# B&R Automation Studio project x20ost (part 4)

#### bnrmytimer.c
```c
/********************************************************************
 * COPYRIGHT -- Kontora
 ********************************************************************
 * Program: bnrmain
 * File: bnrlsens.c
 * Author: Abramenya
 * Created: January 19, 2009
 *******************************************************************/

#include "bnrmytimer.h"
#ifdef _DEFAULT_INCLUDES
 #include <AsDefault.h>
#endif
void CMTimer_OfTimer(This)
{
     DECLARE_MULTI_OPEN(CMTimer,CSystemTimer)
     pB->OfTimer(pB);
}
void CMTimer_OnTimer(This,DWORD dwTime)
{
     DECLARE_MULTI_OPEN(CMTimer,CSystemTimer)
	 pB->OnTimer(pB,dwTime);
	 pT->m_dwSTime = dwTime;
}
void CMTimer_Restart(This)
{
	 DECLARE_MULTI_OPEN(CMTimer,CSystemTimer)
	 pB->OnTimer(pB,pT->m_dwSTime);
}
DWORD CMTimer_GetTime(This)
{
	DECLARE_MULTI_OPEN(CMTimer,CSystemTimer)
	//if pB->m_dwTime
    return pB->m_dwTime;
}
void CMTimer_SetTimer(This,BYTE byFor,BYTE byFrom,BYTE byEvent,BYTE byDir,BYTE bySens,BYTE byBox)
{
     DECLARE_MULTI_OPEN(CMTimer,CSystemTimer)
	 pT->m_byFor   = byFor;
	 pT->m_byFrom  = byFrom;
	 pT->m_byEvent = byEvent;
	 pT->m_byDir   = byDir;
	 pT->m_bySens  = bySens;
	 pT->m_byBox   = byBox;
}
void CMTimer_DoAction(This)
{
	 DECLARE_MULTI_OPEN(CMTimer,CSystemTimer)
	 pT->sMsg.m_swLen        = 9;
	 pT->sMsg.m_sbyFrom      = pT->m_byFrom;
	 pT->sMsg.m_sbyFor       = pT->m_byFor;
	 pT->sMsg.m_sbyIntType   = 0;
	 pT->sMsg.m_sbyServerID  = MYSYSTEM_ID;
	 pT->sMsg.m_sbyDirection = pT->m_byDir;
	 pT->sMsg.m_sbySensor    = pT->m_bySens;
	 pT->sMsg.m_sbyType      = pT->m_byEvent;
	 FPUT(pT->m_byBox,(BYTE*)&pT->sMsg);
}
void CMTimer_CMTimer(This)
{
     DECLARE_MULTI_OPEN(CMTimer,CSystemTimer)
	 DECLARE_REGISTRATION(CMTimer,GetTime)
	 DECLARE_REGISTRATION(CMTimer,OnTimer)
	 DECLARE_REGISTRATION(CMTimer,OfTimer)
	 DECLARE_REGISTRATION(CMTimer,SetTimer)
	 DECLARE_REGISTRATION(CMTimer,Restart)
	 DECLARE_VIRTUAL_FUNC(CMTimer,DoAction)
}
void CMTimer_DCMTimer(This)
{
	 DECLARE_MULTI_OPEN(CMTimer,CSystemTimer)
}
DECLARE_MULTI_CREATE(CMTimer,CSystemTimer)
```

#### bnrobserve.c
```c
/********************************************************************
 * COPYRIGHT -- Kontora
 ********************************************************************
 * Program: bnrmain
 * File: bnrlsens.c
 * Author: Abramenya
 * Created: January 19, 2009
 *******************************************************************/

#include "bnrobserve.h"
#if MYSYSTEM_ID != 5
#ifdef _DEFAULT_INCLUDES
#include <AsDefault.h>
#endif
CObserveModule *pvOBS;
_GLOBAL PFNVOID pfnAnalogDataReq;
_GLOBAL PFNVOID pfnDigitalDataReq;
void AnalogDataReq(void);
void DigitalDataReq(void);
void CObserveModule_Init(This,SSOFTSWITCHTABLE *pSoftSwitchTable)
{
    DECLARE_MULTI_OPEN(CObserveModule,CCyclicSystem)
	pvOBS = pT;
	pfnAnalogDataReq  = AnalogDataReq;
    pfnDigitalDataReq = DigitalDataReq;
	pT->m_byTableVersion = pSoftSwitchTable->byTableVersion;
	strcpy(pT->m_chTableVersionName,pSoftSwitchTable->chTableVersionName);
	pT->m_byAmDirection = pSoftSwitchTable->byAmDirection;
    //#ifdef DEB_CObserveModule
	Info("\n(__)COBSE::>Create Observation Module: %s",pSoftSwitchTable->chTableVersionName);
    //#endif
    pT->CreateObserve(pT,pSoftSwitchTable);
	pT->m_byObsTime = T2SEC;
	InitObject(CMTimer,&pT->m_pRefrechTmr);
	pT->m_pRefrechTmr.SetTimer(&pT->m_pRefrechTmr,MDL_OBSRV,MDL_OBSRV,EV_OBSRV_REFR_TIM_PROC_IND,0,0,DEV_SYSTM_BOX_ID);
}
_GLOBAL INT iCObserveModuleVal;
void CObserveModule_CreateObserve(This,SSOFTSWITCHTABLE *pSoftSwitchTable)
{
    DECLARE_MULTI_OPEN(CObserveModule,CCyclicSystem)
	CDirectionModule *p;
	INT i;
	InitObject(CMFlash,&pT->m_nFlash);
	pT->m_byAmDirection = pSoftSwitchTable->byAmDirection;
	New(sizeof(CDirectionModule*)*pT->m_byAmDirection,pT->m_pDirectionModule);
	for(i=0;i<pT->m_byAmDirection;i++)
	{
	 New(sizeof(CDirectionModule),p);
	 InitObject(CDirectionModule,p);
	 if(p!=NULL)
	 {
	  iCObserveModuleVal++;
	  p->ConnectToComputer(p,pT->m_pComputer);
      p->ConnectToAdmin(p,pT->m_pAdmin);
	  p->m_bySystemID = pT->m_bySystemID;
	  p->Init(p,&pSoftSwitchTable->sDirectionTable[i],&pT->m_nFlash);
	  pT->m_pDirectionModule[i] = p;
	 }
	}
}
void CObserveModule_SetSystemID(This,BYTE bySystemID)
{
     DECLARE_MULTI_OPEN(CObserveModule,CCyclicSystem)
     pT->m_bySystemID = bySystemID;
}
void CObserveModule_ConnectToAdmin(This,CAdmin *pAdmin)
{
     DECLARE_MULTI_OPEN(CObserveModule,CCyclicSystem)
	 pT->m_pAdmin = pAdmin;
}
//_GLOBAL INT nVAL_0;
BOOL CObserveModule_EventHandler(This,SMESSAGE *pMsg)
{
	 BOOL res = TRUE;
     DECLARE_MULTI_OPEN(CObserveModule,CCyclicSystem)
	 CDirectionModule *pD;SPIN sP;CSensor *pS;
	 WORD wValue,wValue1; BYTE byValue,*pBT;
	 #ifdef DEB_CObserveModule
	 if(dwFL&DEB_OUT_OBSR_COMM)
	 Info("\n(%b)COBSE::>MSG::%M",&pT->m_bySystemID,(BYTE*)pMsg);
     #endif
     switch (pMsg->m_sbyFor)
	 {
		case MDL_OBSRV:
             switch (pMsg->m_sbyType)
			 {
                case EV_OBSRV_GET_MODE_REQ: //Запросить выходное состояние сенсоров направления	140
                     if((pD=pT->GetDirection(pT,pMsg->m_sbyDirection))!=0)
					 {
					 pD->GetDirMode(pD,pMsg);
					 #ifdef DEB_CObserveModule
					 if(dwFL&DEB_OUT_OBSR_COMM)
					 Info("\n(%b)COBSE::>DC(%b,X)SET_MODE",&pT->m_bySystemID,&pMsg->m_sbyDirection);
                     #endif
					 }
     	        break;
				case EV_OBSRV_SET_MODE_REQ:
					 if((pD=pT->GetDirection(pT,pMsg->m_sbyDirection))!=0)
					 {
					 pD->SetDirMode(pD,pMsg);
                     #ifdef DEB_CObserveModule
					 if(dwFL&DEB_OUT_OBSR_COMM)
					 Info("\n(%b)COBSE::>DC(%b,X)SET_MODE",&pT->m_bySystemID,&pMsg->m_sbyDirection);
                     #endif
					 }
				break;
				case EV_OBSRV_START_DATA_PROC_REQ:
					 byValue = pMsg->m_sbyInfo[1];
					 pT->m_byObserveProc = pMsg->m_sbyInfo[2];
                     pT->m_byObsTime = byValue;
                     pT->m_pRefrechTmr.OnTimer(&pT->m_pRefrechTmr,pT->m_byObsTime);
					 //pT->m_pRefrechTmr.OnTimer(&pT->m_pRefrechTmr,10);
                     //#ifdef DEB_CObserveModule
					 //if(dwFL&DEB_OUT_OBSR_COMM)
					 //Info("\n(%b)COBSE::>DC(%b,X)START_DATA_PROC_REQ:[%b]:[%b]",&pT->m_bySystemID,&pMsg->m_sbyDirection,&byValue,&pT->m_byObserveProc);
                     //#endif
				break;
				case EV_OBSRV_STOP_DATA_PROC_REQ:
					 pT->m_pRefrechTmr.OfTimer(&pT->m_pRefrechTmr);
                     #ifdef DEB_CObserveModule
					 if(dwFL&DEB_OUT_OBSR_COMM)
					 Info("\n(%b)COBSE::>DC(%b,X)STOP_DATA_PROC_REQ",&pT->m_bySystemID,&pMsg->m_sbyDirection);
                     #endif
				break;
                case EV_OBSRV_REFR_TIM_PROC_IND: //Таймер обновления данных
					 if(pT->m_byObserveProc==0)pT->GetObserveData(pT,EV_OBSRV_GET_OUT_DATA_IND);
					 if(pT->m_byObserveProc==1)pT->GetObserveData(pT,EV_OBSRV_GET_DMC_DATA_IND);
					 //if(pT->m_byObserveProc==0)pfnAnalogDataReq();
					 //if(pT->m_byObserveProc==1)pfnDigitalDataReq();
					 pT->m_pRefrechTmr.OnTimer(&pT->m_pRefrechTmr,pT->m_byObsTime);
					 //pT->m_pRefrechTmr.OnTimer(&pT->m_pRefrechTmr,10);
                     #ifdef DEB_CObserveModule
					 if(dwFL&DEB_OUT_OBSR_COMM)
					 Info("\n(%b)COBSE::>DC(%b,X)GET_INOUT_SDATA_IND",&pT->m_bySystemID,&pMsg->m_sbyDirection);
                     #endif
				break;
				case EV_OBSRV_RFLASH_SAVE_REQ:
				     //nVAL_0++;
					 pT->m_pDirectionModule[0]->m_byDefSett = 0;
			         pT->m_pDirectionModule[0]->Serialize(pT->m_pDirectionModule[0],TRUE);
				break;
                default:
		        break;
			 }
		break;
		case MDL_PSENS://Digital Sensor
			 if((pS=pT->GetSensor(pT,&pD,pMsg->m_sbyDirection,pMsg->m_sbySensor))!=0)
			 pS->EventHandler(pS->pChld,pMsg);
		break;
        #if MYSYSTEM_ID !=4
		case MDL_SENSR:
			 if((pS=pT->GetSensor(pT,&pD,pMsg->m_sbyDirection,pMsg->m_sbySensor))!=0)
			 pS->SEventHandler(pS,pMsg);
		break;
		case MDL_SSENS:
			 if((pS=pT->GetSensor(pT,&pD,pMsg->m_sbyDirection,pMsg->m_sbySensor))!=0)
	         pS->EventHandler(pS->pChld,pMsg);
		break;
        #endif
		case MDL_DIRMD:
			 if((pD=pT->GetDirection(pT,pMsg->m_sbyDirection))!=0)
			 pD->EventHandler(pD,pMsg);
		break;
		default:
		break;
	};
	return res;
}
//_GLOBAL INT nAnData;
void AnalogDataReq(void)
{
	pvOBS->GetObserveData(pvOBS,EV_OBSRV_GET_OUT_DATA_IND);
	//nAnData++;
}
void DigitalDataReq(void)
{
    pvOBS->GetObserveData(pvOBS,EV_OBSRV_GET_DMC_DATA_IND);
}
void CObserveModule_GetObserveData(This,BYTE byEvent)
{
	DECLARE_MULTI_OPEN(CObserveModule,CCyclicSystem)
	INT i,j=0;
	CDirectionModule *p;
	SMESSAGE *pM = &pT->m_nMsg;
	BYTE *pMB = &pM->m_sbyInfo[0];
	pM->m_sbyFrom      = MDL_OBSRV;
	pM->m_sbyFor       = MDL_ARMSY;
	pM->m_sbyIntType   = DEV_ARM_PORT_TCP;
	pM->m_sbyType      = byEvent;
	pM->m_sbyServerID  = pT->m_bySystemID;
	pM->m_sbySensor    = 0xff;
	pM->m_swLen        = 9;
	for(i=0;i<pT->m_byAmDirection;i++)
	{
	 p = pT->m_pDirectionModule[i];
	 if(byEvent==EV_OBSRV_GET_OUT_DATA_IND)j = p->GetXWData(p,(SMESSAGE*)&pMB[j]);
	 if(byEvent==EV_OBSRV_GET_DMC_DATA_IND)j = p->GetDigMcData(p,(SMESSAGE*)&pMB[j]);
	 pM->m_swLen += j;
	 //Info("\n(%b)COBSE::>Put:%w",&pT->m_bySystemID,&pM->m_swLen);
	}
	pM->m_sbyDirection = pT->m_byAmDirection;
	if(pT->m_pAdmin->m_blArmState)
	FPUT(DEV_ARMOT_BOX_ID,(BYTE*)pM);
	if(dwFL&DEB_OUT_OBSR_COMM)
	Info("\n(%b)COBSE::>MSG:%M",&pT->m_bySystemID,(BYTE*)pM);
}
CDirectionModule* CObserveModule_GetDirection(This,BYTE byDir)
{
	DECLARE_MULTI_OPEN(CObserveModule,CCyclicSystem)
	CDirectionModule *pD;
	if(byDir<pT->m_byAmDirection)
		return pD = pT->m_pDirectionModule[byDir];
	return 0;
}
CSensor* CObserveModule_GetSensor(This,CDirectionModule **pD,BYTE byDir,BYTE bySensor)
{
	DECLARE_MULTI_OPEN(CObserveModule,CCyclicSystem)
	CDirectionModule *pDM = *pD;
	if(byDir<pT->m_byAmDirection)
	{
	 pDM = pT->m_pDirectionModule[byDir];
	 *pD = pDM;
	 if(bySensor < pDM->m_byAmSwitching)
	 return pDM->m_pSensor[bySensor];
	}
	return 0;
}
void CObserveModule_CyclicProc(This)
{
	DECLARE_MULTI_OPEN(CObserveModule,CCyclicSystem)
	CDirectionModule *p;INT i;
    for(i=0;i<pT->m_byAmDirection;i++)
	{
	  p = pT->m_pDirectionModule[i];
	  p->ObserveProc(p);
	}
}
void CObserveModule_ConnectToComputer(This,CComputer *pComputer)
{
    DECLARE_MULTI_OPEN(CObserveModule,CCyclicSystem)
	pT->m_pComputer = pComputer;
}
void CObserveModule_CObserveModule(This)
{
    DECLARE_MULTI_OPEN(CObserveModule,CCyclicSystem)
	DECLARE_REGISTRATION(CObserveModule,Init)
	DECLARE_REGISTRATION(CObserveModule,ConnectToComputer)
	DECLARE_REGISTRATION(CObserveModule,CreateObserve)
	DECLARE_REGISTRATION(CObserveModule,GetObserveData)
	DECLARE_REGISTRATION(CObserveModule,SetSystemID)
	DECLARE_REGISTRATION(CObserveModule,GetDirection)
	DECLARE_REGISTRATION(CObserveModule,GetSensor)
	DECLARE_REGISTRATION(CObserveModule,SetSystemID)
	DECLARE_REGISTRATION(CObserveModule,ConnectToAdmin)
	DECLARE_VIRTUAL_FUNC(CObserveModule,EventHandler)
	DECLARE_VIRTUAL_FUNC(CObserveModule,CyclicProc)
}
void CObserveModule_DCObserveModule(This)
{
	DECLARE_MULTI_OPEN(CObserveModule,CCyclicSystem)
	BYTE i;
	for(i=0;i<pT->m_byAmDirection;i++)
	DestroyObject(CDirectionModule,pT->m_pDirectionModule[i]);
	Delete(sizeof(CDirectionModule*)*pT->m_byAmDirection,pT->m_pDirectionModule);
}
DECLARE_MULTI_CREATE(CObserveModule,CCyclicSystem)
#endif
```

#### bnroutgate.c
```c
/********************************************************************
 * COPYRIGHT -- Kontora
 ********************************************************************
 * Program: bnrmain
 * File: bnrlsens.c
 * Author: Abramenya
 * Created: January 19, 2009
 *******************************************************************/

#include "bnroutgate.h"
#ifdef _DEFAULT_INCLUDES
 #include <AsDefault.h>
#endif
#if MYSYSTEM_ID != 5
void COutGate_Init(This,BYTE byID,BYTE byType,BYTE byOType,BYTE byMode,REAL rMinRamp,REAL rMaxRamp,CPin *pPin,UINT wLo,UINT wHi,UINT wIni,BYTE byState,WORD wBase,WORD wOTime,SINT *pName)
{
    DECLARE_SINGLE_OPEN(COutGate)
	REAL rHL        = (REAL)(wHi-wLo);
	REAL rIP        = (REAL)wIni;
	pT->m_rMinRamp  = rMinRamp;
	pT->m_rMaxRamp  = rMaxRamp;
	pT->m_wBase     = wBase;
	pT->m_byState   = byState;
	pT->m_byGateID  = byID;
	pT->m_byType    = byType;
	pT->m_byOType   = byOType;  //BASE_GTE
	pT->m_byMode    = byMode;
	pT->m_wQTime    = SYSTEM_QTIME;
	pT->m_wLoLimit  = 0;
	pT->m_wHiLimit  = wHi-wLo;
    pT->m_wIniState = (UINT)(rHL*rIP/100.0);
	pT->m_wCurrOpenState = pT->m_wIniState;
	pT->m_dwTime    = 0;
	pT->m_pConnectionPin = pPin;
	if(pPin!=0)pT->m_pwOut = (UINT*)pPin->GetAddrPin(pPin->pChld); else
	pT->m_pwOut = &pT->m_wOut;
	pT->m_wTick     = 0;
	pT->m_wOTime = wOTime;
	if(pT->m_wOTime==0) pT->m_wOTime=1;
	pT->m_wMaxQt = (REAL)pT->m_wOTime*10;
	pT->m_wTickConst = (REAL)pT->m_wHiLimit/pT->m_wMaxQt;
    pT->m_wTickOpen  = pT->m_wTickConst;
	pT->m_blProccState = FALSE;
	pT->m_wMinRampValue = (UINT)(rHL*pT->m_rMinRamp);
	pT->m_wMaxRampValue = (UINT)(rHL*pT->m_rMaxRamp);

	strcpy(pT->m_chName,pName);
}
void COutGate_SetOutTime(This,WORD wValue)
{
    DECLARE_SINGLE_OPEN(COutGate)
	pT->m_wMaxQt = (REAL)wValue*10;
	if(pT->m_wMaxQt==0)return;
    pT->m_wTickConst = pT->m_wHiLimit/pT->m_wMaxQt;
	pT->m_wTickOpen  = pT->m_wTickConst;
}
void COutGate_SetHiLimit(This,WORD wValue)
{
    DECLARE_SINGLE_OPEN(COutGate)
    pT->m_wHiLimit = wValue;
	pT->m_wTickConst = pT->m_wHiLimit/pT->m_wMaxQt;
    pT->m_wTickOpen  = pT->m_wTickConst;
}
//UINT _GLOBAL nmMaxRamp,nOutVal,nMinR,nMaxR,nCOpen;
//REAL _GLOBAL rgValue,rHILM,rMaxRamp;
void COutGate_SetMinRamp(This,REAL rValue)
{
    DECLARE_SINGLE_OPEN(COutGate)
	REAL rMaxValue = (REAL)pT->m_wHiLimit;
    pT->m_rMinRamp = rValue;
	pT->m_wMinRampValue = (UINT)(rMaxValue*pT->m_rMinRamp);
}
void COutGate_SetMaxRamp(This,REAL rValue)
{
    DECLARE_SINGLE_OPEN(COutGate)
	REAL rMaxValue = (REAL)pT->m_wHiLimit;
	pT->m_rMaxRamp = rValue;
	pT->m_wMaxRampValue = (UINT)(rMaxValue*pT->m_rMaxRamp);

	//nmMaxRamp = pT->m_wHiLimit;
	//rHILM     = rMaxValue;
	//rgValue   = rValue;
	//rMaxRamp  = pT->m_wMaxRampValue;
}
void COutGate_OpenGate(This,REAL rOpenState)
{
    DECLARE_SINGLE_OPEN(COutGate)
	UINT wEndState;
	REAL rHi;
	//if(!pT->m_blProccState)
	{
	 rHi = (REAL)pT->m_wHiLimit;
	 wEndState = (UINT)(rOpenState*rHi/100.0);
	 if (wEndState==pT->m_wCurrOpenState) return;
	 pT->m_wTickOpen = pT->m_wTickConst;
	 if (wEndState < pT->m_wCurrOpenState)
     pT->m_wTickOpen = -pT->m_wTickConst;
     pT->m_wTick = (DWORD)(abs(pT->m_wCurrOpenState-wEndState)/pT->m_wTickConst);
	 pT->m_wOperGate = (REAL)pT->m_wCurrOpenState;
	 pT->m_blProccState = TRUE;
	};
}
void COutGate_OpenGateReq(This,BYTE byOpenState)
{
    DECLARE_SINGLE_OPEN(COutGate)
	UINT wEndState;
	REAL rHi;
	if (byOpenState<=100)
	{
	 rHi = (REAL)pT->m_wHiLimit;
     wEndState = (UINT)((REAL)byOpenState*rHi/100.0);
	 pT->SetManGate(pT,wEndState);
	}
}
void COutGate_StopGate(This)
{
    DECLARE_SINGLE_OPEN(COutGate)
    pT->m_blProccState = FALSE;
	pT->m_wTick = 0;
}
void COutGate_SetGate(This,UINT wValue)
{
	DECLARE_SINGLE_OPEN(COutGate)
	//nOutVal = wValue;
	//nMinR   = pT->m_wMinRampValue;
	//nMaxR   = pT->m_wMaxRampValue;
	if (wValue<pT->m_wMinRampValue) wValue = pT->m_wMinRampValue;
	if (wValue>pT->m_wMaxRampValue) wValue = pT->m_wMaxRampValue;
	//if((wValue>=pT->m_wMinRampValue)&&(wValue<=pT->m_wMaxRampValue+20))
	//{
	pT->m_wCurrOpenState = wValue;
	//nCOpen = wValue;
    if(pT->m_byState==ST_OPEN)
	{
	 if(pT->m_byOType==NZ) *pT->m_pwOut = pT->m_wBase+pT->m_wCurrOpenState;
	 if(pT->m_byOType==NO) *pT->m_pwOut = pT->m_wBase+(pT->m_wHiLimit-pT->m_wCurrOpenState);
	}
	//}
}
void COutGate_SetManGate(This,UINT wValue)
{
	DECLARE_SINGLE_OPEN(COutGate)
	pT->m_wCurrOpenState = wValue;
    if(pT->m_byState==ST_OPEN)
	{
	 if(pT->m_byOType==NZ) *pT->m_pwOut = pT->m_wBase+pT->m_wCurrOpenState;
	 if(pT->m_byOType==NO) *pT->m_pwOut = pT->m_wBase+(pT->m_wHiLimit-pT->m_wCurrOpenState);
	}
}
UINT COutGate_GetGate(This)
{
	DECLARE_SINGLE_OPEN(COutGate)
	if(pT->m_byOType==NZ)return pT->m_wBase+pT->m_wCurrOpenState;
	if(pT->m_byOType==NO)return pT->m_wBase+(pT->m_wHiLimit-pT->m_wCurrOpenState);
	return 0;
}
BYTE COutGate_GetPrcGate(This)
{
	DECLARE_SINGLE_OPEN(COutGate)
	//REAL rC = pT->m_wCurrOpenState;
	//REAL rH = pT->m_wHiLimit;
	//return (BYTE)(100.0*rC/rH);
	return (BYTE)(100.0*pT->m_wCurrOpenState/pT->m_wHiLimit);
	//return (BYTE)(100.0*pT->m_wCurrOpenState/6683.0);
}
void COutGate_RunGate(This)
{
    DECLARE_SINGLE_OPEN(COutGate)
	if(pT->m_blProccState)
	{
	 if(pT->m_wTick!=0)
	 {
	  pT->m_wOperGate += pT->m_wTickOpen;
	  //Info("\n(__)Tick:%b Val:%w",&pT->m_wTick,&pT->m_wCurrOpenState.iValue);
	  pT->SetManGate(pT,(UINT)pT->m_wOperGate);
	  pT->m_wTick--;
	 }else pT->m_blProccState = FALSE;
	}
}
void COutGate_SetDefault(This)
{
    DECLARE_SINGLE_OPEN(COutGate)
	pT->SetGate(pT,pT->m_wIniState);
}
void COutGate_SetState(This,BYTE byState)
{
    DECLARE_SINGLE_OPEN(COutGate)
	if(byState==ST_INIT)pT->SetDefault(pT);
	pT->m_byState = byState;
}
void COutGate_COutGate(This)
{
    DECLARE_SINGLE_OPEN(COutGate)
	DECLARE_REGISTRATION(COutGate,Init)
	DECLARE_REGISTRATION(COutGate,OpenGate)
    DECLARE_REGISTRATION(COutGate,SetGate)
	DECLARE_REGISTRATION(COutGate,GetGate)
	DECLARE_REGISTRATION(COutGate,RunGate)
	DECLARE_REGISTRATION(COutGate,SetDefault)
	DECLARE_REGISTRATION(COutGate,SetState)
	DECLARE_REGISTRATION(COutGate,GetPrcGate)
	DECLARE_REGISTRATION(COutGate,SetMinRamp)
	DECLARE_REGISTRATION(COutGate,SetMaxRamp)
	DECLARE_REGISTRATION(COutGate,SetHiLimit)
	DECLARE_REGISTRATION(COutGate,SetManGate)
	DECLARE_REGISTRATION(COutGate,StopGate)
	DECLARE_REGISTRATION(COutGate,SetOutTime)
	DECLARE_REGISTRATION(COutGate,OpenGateReq)
}
void COutGate_DCOutGate(This)
{
	DECLARE_SINGLE_OPEN(COutGate)
}
DECLARE_SINGLE_CREATE(COutGate)
#endif
```

#### bnrpin.c
```c
/********************************************************************
 * COPYRIGHT -- Kontora
 ********************************************************************
 * Program: bnrmain
 * File: bnrlsens.c
 * Author: Abramenya
 * Created: January 19, 2009
 *******************************************************************/

#include "bnrpin.h"
#ifdef _DEFAULT_INCLUDES
 #include <AsDefault.h>
#endif
#ifdef DEB_CPin
SINT *chPinState[] =
{
	"DEF",
	"ONN",
	"OFF",
	"TRI",
};
SINT *chPinType[] =
{
	"DEFAULT_PIN",
	"AN_INOT_INT",
	"DG_INOT_BOL",
	"ST_INPT_USI",
	"ST_OUTP_USI"
};
#endif
void CPin_Init(This,SHARDPIN*pPin,SHARDPIN *pAlPin)
{
    DECLARE_SINGLE_OPEN(CPin)
	pT->m_pvAlmState  = pAlPin->pvValue;
	pT->m_byPinState  = pPin->byPinState;
	pT->m_byPinNumber = pPin->byPinNumber;
	pT->InitPin(pC,pPin->pvValue);
	pT->m_blPinON  = FALSE;
	pT->m_blPinOFF = FALSE;
    #ifdef DEB_CPin
	Info("\n(%b)CPINS::>Create Pin: State:[%s] Type:[%s]",&pPin->byPinNumber,chPinState[pPin->byPinState],chPinType[pPin->byPinType]);
    #endif
}

void CPin_SetSlot(This,BYTE bySlot)
{
	DECLARE_SINGLE_OPEN(CPin)
    pT->m_bySlotNumber = bySlot;
}
PVOID CPin_GetAddrPin(This)
{
	DECLARE_SINGLE_OPEN(CPin)
	return 0;
}
BYTE CPin_GetState(This)
{
    DECLARE_SINGLE_OPEN(CPin)
	SPIN sP;
	pT->GetPin(pC,&sP);
	if(sP.blValue)
	{
	 if(pT->m_blPinON==FALSE)
	 {
	  pT->m_blPinON = TRUE;
	  pT->m_blPinOFF= FALSE;
	  return PIN_STATE_ONN;
	 }else return PIN_STATE_TRI;
	}else
	{
	 if(pT->m_blPinOFF==FALSE)
	 {
	  pT->m_blPinOFF= TRUE;
	  pT->m_blPinON = FALSE;
	  return PIN_STATE_OFF;
	 }else return PIN_STATE_TRI;
	}
}
void CPin_GetPin(This,SPIN *sP)
{
    DECLARE_SINGLE_OPEN(CPin)
}
void CPin_CPin(This)
{
    DECLARE_SINGLE_OPEN(CPin)
	DECLARE_REGISTRATION(CPin,Init)
	DECLARE_REGISTRATION(CPin,SetSlot)
	DECLARE_REGISTRATION(CPin,GetAddrPin)
	DECLARE_REGISTRATION(CPin,GetPin)
	DECLARE_REGISTRATION(CPin,GetState)
}
void CPin_DCPin(This)
{
	DECLARE_SINGLE_OPEN(CPin)
}
DECLARE_SINGLE_CREATE(CPin)
```

#### bnrpob.c
```c
#include "bnrpob.h"
#include "bnrmessage.h"
#ifndef WIN32
_GLOBAL pBOX pBufferHiLev[MAXNAMEBUF];
_GLOBAL pBOX nMirrorBuffer;
_GLOBAL BOOL blSMB;
#else
pBOX pBufferHiLev[MAXNAMEBUF];
pBOX nMirrorBuffer;
BOOL blSMB;
#endif
void FFREE(BYTE b_lNmBox)
{
	pBOX *p;
	if(b_lNmBox>MAXNAMEBUF) return;
	nMirrorBuffer.pb_mBoxCont = 0;
	nMirrorBuffer.w_mBoxMesCt = 1;
	blSMB = FALSE;
	p = &pBufferHiLev[b_lNmBox];
	p->w_mBoxSize  = p->w_mBoxCSize;
    p->w_mBoxWrite = 0;
    p->w_mBoxRead  = 0;
    p->w_mBoxMesCt = 0;
}
void FINIT(void)
{
	//BYTE i;
	//for(i=0;i<MAXNAMEBUF-1;i++)pBufferHiLev[i].pb_mBoxCont = 1;
}
int FDEFINE(BYTE b_lNmBox,WORD w_lBoxSize)
{
	pBOX *p;
    if(b_lNmBox>MAXNAMEBUF) return NULL;
	p = &pBufferHiLev[b_lNmBox];
	//if(p->pb_mBoxCont!=1) return b_lNmBox;
	New(sizeof(BYTE)*(w_lBoxSize+BOX_TRANS_SIZE),p->pb_mBoxCont);
    if(p==NULL) return NULL;
	p->w_mBoxSize  = w_lBoxSize;
    p->w_mBoxCSize = w_lBoxSize;
    p->w_mBoxWrite = 0;
    p->w_mBoxRead  = 0;
    p->w_mBoxMesCt = 0;
    #ifdef DEF_CRT_BOX
	Info("\n(%b)CSBOX::>Create System Box.Size:%w",&b_lNmBox,&pBufferHiLev[b_lNmBox]->w_mBoxCSize);
    //Info("\n(%b)CRT:BOX:>:AD[%a]:WR[%w]:RD[%w]:SZ[%w]:CT[%w]",&b_lNmBox,&p,&p->w_mBoxWrite,&p->w_mBoxRead,&p->w_mBoxSize,&p->w_mBoxMesCt);
    #endif
    return 1;
}
void FDELETE(BYTE b_lNmBox)
{
	pBOX *p;
	p = &pBufferHiLev[b_lNmBox];
    Delete(p->w_mBoxCSize+BOX_TRANS_SIZE,p->pb_mBoxCont);
    p->pb_mBoxCont = 0;
    #ifdef DEF_CRT_BOX
    Info("\n(%b)DEL:BOX",&b_lNmBox);
    #endif
}
int FCHECK(BYTE b_lNmBox)
{
    return pBufferHiLev[b_lNmBox].w_mBoxMesCt;
}
int FCHECKM(BYTE b_lNmBox)
{
	if(!blSMB)
	{
	 memcpy(&nMirrorBuffer,&pBufferHiLev[b_lNmBox],sizeof(pBOX));
	 blSMB = TRUE;
	}
    return nMirrorBuffer.w_mBoxMesCt;
}
int FPUT(BYTE b_lNmBox,BYTE *pb_lInBox)
{
	pBOX *p;
    WORD w_lLength;
	p = &pBufferHiLev[b_lNmBox];
    w_lLength = *(WORD*)pb_lInBox;
    if(!p->pb_mBoxCont)return 0;
    if((w_lLength>p->w_mBoxSize)||(w_lLength<2))return 0;
	memcpy(&p->pb_mBoxCont[p->w_mBoxWrite],pb_lInBox,w_lLength);
    p->w_mBoxWrite += w_lLength;
    p->w_mBoxSize  -= w_lLength;
    p->w_mBoxMesCt ++;
    if(p->w_mBoxWrite>p->w_mBoxCSize) p->w_mBoxWrite = 0;
    #ifdef DEF_INF_BOX
    Info("\n(%b)PUTB:>:LN[%w]:WR[%w]:RD[%w]:SZ[%w]:CT[%w]",&b_lNmBox,&w_lLength,&p->w_mBoxWrite,&p->w_mBoxRead,&p->w_mBoxSize,&p->w_mBoxMesCt);
    #endif
    #ifdef DEF_PUT_BOX
    Info("\n(%b)PUTB[%w]:>:%m",&b_lNmBox,&p->w_mBoxMesCt,pb_lInBox);
    #endif
    return 1;
}
int FPUT1(BYTE b_lNmBox,BYTE *pb_lInBox)
{
	if(FPUT(b_lNmBox,pb_lInBox)==0)
	{
     FFREEM(b_lNmBox);
	 if(FPUT(b_lNmBox,pb_lInBox)==0)
	 return 0;
	}
	return 1;
}
int FFREEM(BYTE b_lNmBox)
{
    pBOX *p;
	BYTE *pb_lLength;
	WORD  wLng;
    p = &pBufferHiLev[b_lNmBox];
	if(!p->pb_mBoxCont)return 0;
	if(!p->w_mBoxMesCt)return 0;
    pb_lLength = (BYTE*)&p->pb_mBoxCont[p->w_mBoxRead];
    #ifdef WIN32
	wLng = (((WORD)pb_lLength[1])<<8)|(WORD)pb_lLength[0];
    #else
	wLng = (((WORD)pb_lLength[0])<<8)|(WORD)pb_lLength[1];
    #endif
    //memcpy(pb_lInBox,pb_lLength,wLng);
    p->w_mBoxRead += wLng;
    p->w_mBoxSize += wLng;
    p->w_mBoxMesCt --;
    if(p->w_mBoxRead>p->w_mBoxCSize) p->w_mBoxRead = 0;
    return 1;
}
void FSMRB(BYTE b_lNmBox)
{
    memcpy(&nMirrorBuffer,&pBufferHiLev[b_lNmBox],sizeof(pBOX));
	blSMB = FALSE;
}
int FGET1(BYTE b_lNmBox,BYTE *pb_lInBox)
{
	pBOX *p;
	BYTE *pb_lLength;
	WORD  wLng;
	p = &nMirrorBuffer;
	if(!p->pb_mBoxCont)return 0;
	if(!p->w_mBoxMesCt)return 0;
    pb_lLength = (BYTE*)&p->pb_mBoxCont[p->w_mBoxRead];
    #ifdef WIN32
	wLng = (((WORD)pb_lLength[1])<<8)|(WORD)pb_lLength[0];
    #else
	wLng = (((WORD)pb_lLength[0])<<8)|(WORD)pb_lLength[1];
    #endif
    memcpy(pb_lInBox,pb_lLength,wLng);
    p->w_mBoxRead += wLng;
    p->w_mBoxSize += wLng;
    p->w_mBoxMesCt --;
    if(p->w_mBoxRead>p->w_mBoxCSize) p->w_mBoxRead = 0;
    return 1;
}
int FGET(BYTE b_lNmBox,BYTE *pb_lInBox)
{
    pBOX *p;
	BYTE *pb_lLength;
	WORD  wLng;
    p = &pBufferHiLev[b_lNmBox];
	if(!p->pb_mBoxCont)return 0;
	if(!p->w_mBoxMesCt)return 0;
    pb_lLength = (BYTE*)&p->pb_mBoxCont[p->w_mBoxRead];
    #ifdef WIN32
	wLng = (((WORD)pb_lLength[1])<<8)|(WORD)pb_lLength[0];
    #else
	wLng = (((WORD)pb_lLength[0])<<8)|(WORD)pb_lLength[1];
    #endif
    memcpy(pb_lInBox,pb_lLength,wLng);
    p->w_mBoxRead += wLng;
    p->w_mBoxSize += wLng;
    p->w_mBoxMesCt --;
    if(p->w_mBoxRead>p->w_mBoxCSize) p->w_mBoxRead = 0;
    #ifdef DEF_INF_BOX
    Info("\n(%b)GETB:>:LN[%w]:WR[%w]:RD[%w]:SZ[%w]:CT[%w]",&b_lNmBox,(WORD*)pb_lLength,&p->w_mBoxWrite,&p->w_mBoxRead,&p->w_mBoxSize,&p->w_mBoxMesCt);
    #endif
    #ifdef DEF_GET_BOX
    Info("\n(%b)GETB[%w]:>:%m",&b_lNmBox,&p->w_mBoxMesCt,pb_lInBox);
    #endif
    return 1;
}
```

#### bnrprocmanager.c
```c
/********************************************************************
 * COPYRIGHT -- Kontora
 ********************************************************************
 * Program: bnrmain
 * File: bnrlsens.c
 * Author: Abramenya
 * Created: January 19, 2009
 *******************************************************************/

#include "bnrprocmanager.h"
#ifdef _DEFAULT_INCLUDES
 #include <AsDefault.h>
#endif
#ifdef DEB_CProcManager
SINT *chManState[] =
{
	"ONN",
    "OFF",
};
#endif
void CProcManager_Init(This,DWORD dwTicTime,BOOL blStatistic)
{
	 INT i;
     DECLARE_SINGLE_OPEN(CProcManager)
	 for(i=0;i<DEV_MAX_CYC_PROC;i++)
	 pT->m_nCyclicSystem[i] = NULL;
     for(i=0;i<DEV_MAX_SYS_TIMR;i++)
	 pT->m_nSystemTimer[i] = NULL;
	 pT->m_iProcCounter = 0;
	 pT->m_dwTicTime = dwTicTime;
	 pT->m_nMaxProc = 0;
	 pT->m_byCheckQuant = 0;
	 pT->m_nMaxTimer = 0;
	 pT->m_blStatistic = blStatistic;
     #ifdef DEB_CProcManager
	 Info("\n(__)CPMAN::>Create Process Manager:State:%s ",chManState[pT->m_blState]);
     #endif
}
void CProcManager_SetTicTime(This,DWORD dwTicTime)
{
     DECLARE_SINGLE_OPEN(CProcManager)
	 pT->m_dwTicTime = dwTicTime;
}
BOOL CProcManager_ConnectTimer(This,CSystemTimer *pSTimer)
{
	BYTE i;
	DECLARE_SINGLE_OPEN(CProcManager)
	for(i=0;i<DEV_MAX_SYS_TIMR;i++)
	{
	  if(pT->m_nSystemTimer[i]==NULL)
	  {
        pT->m_nSystemTimer[i] = pSTimer;
		pT->m_nSystemTimer[i]->SetTimerID(pT->m_nSystemTimer[i],i);
		pT->m_nMaxTimer++;
		return TRUE;
	  }
	}
	return FALSE;
}
BOOL CProcManager_DisconnectTimer(This,CSystemTimer *pSTimer)
{
	int i;
	DECLARE_SINGLE_OPEN(CProcManager)
	CSystemTimer *p;
	for(i=0;i<pT->m_nMaxTimer;i++)
	{
	 p = pT->m_nSystemTimer[i];
	 if(p!=NULL)
	 {
	  if(p->m_byTimerID==i)
	  {
       p = NULL;
	   if(pT->m_nMaxTimer>0)pT->m_nMaxTimer--;
	   return TRUE;
	  }
	 }
	}
	return FALSE;
}
BOOL CProcManager_ConnectProc(This,CCyclicSystem *pCSystem)
{
	 int i;
     DECLARE_SINGLE_OPEN(CProcManager)
	 for(i=0;i<DEV_MAX_CYC_PROC;i++)
	 {
       if(pT->m_nCyclicSystem[i]==NULL)
	   {
         pT->m_nCyclicSystem[i] = pCSystem;
		 pT->m_nMaxProc++;
		 return TRUE;
	   }
	 }
	 return FALSE;
}
void CProcManager_DeleteProc(This,SINT *chName)
{
	 INT iIndex;
     DECLARE_SINGLE_OPEN(CProcManager)
	 if((iIndex=pT->Find(pT,chName))==-1)
	 {
	   pT->m_nCyclicSystem[iIndex] = NULL;
	   if(pT->m_nMaxProc>0)pT->m_nMaxProc--;
	 }
}
int CProcManager_Find(This,SINT *chName)
{
	 INT i;
     DECLARE_SINGLE_OPEN(CProcManager)
	 for(i=0;i<DEV_MAX_CYC_PROC;i++)
	 {
	  if(strcmp(pT->m_nCyclicSystem[i]->m_chProcName,chName)==0)
	     return i;
	 }
	 return -1;
}
void CProcManager_SuspendThread(This,SINT *chName)
{
	 INT iIndex;
	 CCyclicSystem *p;
     DECLARE_SINGLE_OPEN(CProcManager)
	 if((iIndex=pT->Find(pT,chName))==-1)
	 {
	  p = pT->m_nCyclicSystem[iIndex];
	  p->SetState(p,DEV_CJOB_ST_SUSP);
	 }
}
void CProcManager_ResumeThread(This,SINT *chName)
{
	INT iIndex;
	CCyclicSystem *p;
	DECLARE_SINGLE_OPEN(CProcManager)
	if((iIndex=pT->Find(pT,chName))==-1)
	{
	 p = pT->m_nCyclicSystem[iIndex];
	 p->SetState(p,DEV_CJOB_ST_RESM);
	}
}
void CProcManager_SuspendAll(This)
{
	int i;
	CCyclicSystem *p;
	DECLARE_SINGLE_OPEN(CProcManager)
	for(i=0;i<DEV_MAX_CYC_PROC;i++)
	{
     p = pT->m_nCyclicSystem[i];
	 if(p!=NULL)
  	 p->SetState(p,DEV_CJOB_ST_SUSP);
	}
}
void CProcManager_ResumeAll(This)
{
	int i;
	CCyclicSystem *p;
	DECLARE_SINGLE_OPEN(CProcManager)
	for(i=0;i<DEV_MAX_CYC_PROC;i++)
	{
	 p = pT->m_nCyclicSystem[i];
	 if(p!=NULL)
	 p->SetState(p,DEV_CJOB_ST_RESM);
	}
}
//_GLOBAL INT nProc00;
void CProcManager_Run(This)
{
	 INT i;
	 CCyclicSystem *p;
	 CSystemTimer *pS;
     DECLARE_SINGLE_OPEN(CProcManager)
	 //Proc Section
     if(pT->m_blState == DEV_PROC_STT_ONN)
	 {
     for(i=0;i<pT->m_nMaxProc;i++)
     {
	  p = pT->m_nCyclicSystem[i];
	  //if (p!=NULL)
      if ((pT->m_iProcCounter%p->m_byPeriod)==0)
      if(p->m_byStateProc==DEV_CJOB_ST_RESM)
	  {
      p->CyclicProc(p->pChld);
	  p->GetMessage(p);
	  }
     }
	 }
     //Timer Section
	 if(pT->m_iProcCounter%2==0)
	 {
	 //nProc00++;
	 for(i=0;i<pT->m_nMaxTimer;i++){pS = pT->m_nSystemTimer[i];pS->RunTimer(pS);}
	 }
	 pT->m_iProcCounter++;

	 //Info("\nTime[%w]",&pT->m_iProcCounter);
	 //if(dwFL&DEB_OUT_PMAN_STAT)
	 //if (pT->m_iProcCounter%PRC_MAN_CH_QUANT==0) pT->GetTimeStatistic(pT);
}
void CProcManager_GetTimeStatistic(This)
{
     DECLARE_SINGLE_OPEN(CProcManager)
	 INT i;
	 CCyclicSystem *p;
	 DWORD dwTime;
	 for(i=0;i<pT->m_nMaxProc;i++)
     {
	   p = pT->m_nCyclicSystem[i];
	   dwTime = p->m_dwAmoutQuant*pT->m_dwTicTime;
	   #ifdef DEB_CProcManager
	   Info("\n(%b)CPMAN::>Tic: %d.Time: %d.Proc: %s",&pT->m_byCheckQuant,&p->m_dwAmoutQuant,&dwTime,p->m_chProcName);
	   #endif
	 }
	 pT->m_byCheckQuant++;
}
void CProcManager_Start(This)
{
     DECLARE_SINGLE_OPEN(CProcManager)
     pT->m_blState = DEV_PROC_STT_ONN;
     #ifdef DEB_CProcManager
	 Info("\n(__)CPMAN::>Start Process Manager");
     #endif
}
void CProcManager_Stop(This)
{
     DECLARE_SINGLE_OPEN(CProcManager)
     pT->m_blState = DEV_PROC_STT_OFF;
     #ifdef DEB_CProcManager
	 Info("\n(__)CPMAN::>Stop Process Manager");
     #endif
}
void CProcManager_CProcManager(This)
{
     DECLARE_SINGLE_OPEN(CProcManager)
	 DECLARE_REGISTRATION(CProcManager,Init)
	 DECLARE_REGISTRATION(CProcManager,ConnectProc)
	 DECLARE_REGISTRATION(CProcManager,ConnectTimer)
	 DECLARE_REGISTRATION(CProcManager,DisconnectTimer)
     DECLARE_REGISTRATION(CProcManager,DeleteProc)
	 DECLARE_REGISTRATION(CProcManager,SuspendThread)
     DECLARE_REGISTRATION(CProcManager,ResumeThread)
	 DECLARE_REGISTRATION(CProcManager,SuspendAll)
	 DECLARE_REGISTRATION(CProcManager,ResumeAll)
	 DECLARE_REGISTRATION(CProcManager,Find)
	 DECLARE_REGISTRATION(CProcManager,Run)
	 DECLARE_REGISTRATION(CProcManager,Start)
	 DECLARE_REGISTRATION(CProcManager,Stop)
	 DECLARE_REGISTRATION(CProcManager,SetTicTime)
	 DECLARE_REGISTRATION(CProcManager,GetTimeStatistic)
	 pT->m_blState = DEV_PROC_STT_OFF;
}
void CProcManager_DCProcManager(This)
{
	DECLARE_SINGLE_OPEN(CProcManager)
}
DECLARE_SINGLE_CREATE(CProcManager)
```

#### bnrregedit.c
```c
/********************************************************************
 * COPYRIGHT -- Kontora
 ********************************************************************
 * Program: bnrmain
 * File: bnrlsens.c
 * Author: Abramenya
 * Created: January 19, 2009
 *******************************************************************/

#include "bnrregedit.h"
#ifdef _DEFAULT_INCLUDES
 #include <AsDefault.h>
#endif
extern SSOFTSWITCHTABLE nSoftSwitchTable;
extern SHARDCOMPUTERTABLE nConfigTable;
void CRegModule_Init(This)
{
    DECLARE_SINGLE_OPEN(CRegModule)
	SREGADDR nA;
	nA.byA0 = 0;
	nA.byA1 = 0;
	nA.byA2 = 0;
	FDEFINE(BOX_REG,BOX_REG_SZ);
	pT->m_pSCT = &nSoftSwitchTable;
    pT->m_pHCT = &nConfigTable;
	//pT->CreateKpParam(pT,&nA);
	//pT->CreatePortParam(pT,&nA);
	//pT->CreateHardParam(pT,&nA);
	//pT->CreateSoftParam(pT,&nA);
	//pT->SetKpParam(pT,&nA);
}

BYTE CRegModule_QueryParam(This,SREGADDR *pA)
{
    DECLARE_SINGLE_OPEN(CRegModule)
	switch(pA->byA0)
	{
	  case REG_KPPAR_ADDR:
		   return pT->CreateKpParam(pT,pA);
	  case REG_PORTT_ADDR:
		   return pT->CreatePortParam(pT,pA);
	  case REG_HARDT_ADDR:
		   return pT->CreateHardParam(pT,pA);
	  case REG_SOFTI_ADDR:
		   return pT->CreateSoftTIParam(pT,pA);
	  case REG_SOFTS_ADDR:
		   return pT->CreateSoftTSParam(pT,pA);
	  case REG_SOFTU_ADDR:
		   return pT->CreateSoftTUParam(pT,pA);
	  case REG_SOFTR_ADDR:
		   return pT->CreateSoftTRParam(pT,pA);
	}
	return 0;
}
BYTE CRegModule_SaveParam(This,SREGPARAM *pA)
{
    DECLARE_SINGLE_OPEN(CRegModule)
	switch(pA->byA0)
	{
	  case REG_KPPAR_ADDR:
		   return pT->SetKpParam(pT,pA);
	  case REG_PORTT_ADDR:
		   return pT->SetPortParam(pT,pA);
	  case REG_HARDT_ADDR:
		   return pT->SetHardParam(pT,pA);
	  case REG_SOFTI_ADDR:
		   return pT->SetSoftTIParam(pT,pA);
	  case REG_SOFTS_ADDR:
		   return pT->SetSoftTSParam(pT,pA);
	  case REG_SOFTU_ADDR:
		   return pT->SetSoftTUParam(pT,pA);
	  case REG_SOFTR_ADDR:
		   return pT->SetSoftTRParam(pT,pA);
	  default:
	  return 0;
	}
}
BYTE CRegModule_CreateKpParam(This,SREGADDR *pA)
{
    DECLARE_SINGLE_OPEN(CRegModule)
	BYTE i;
	SREGPARAM sP;
	BYTE *pM = (BYTE*)&sP;
	SKPPARAM *pH = pT->m_pHCT->pKpParam;
	FFREE(BOX_REG);
    sP.wSize  = sizeof(SREGPARAM);
	sP.byA0   = pA->byA0;
	sP.byA1   = pA->byA1;
	//if(sP.byA1==0xff)
    if(pA->byA1==0){sP.byA2 = 0;for(i=0;i<8;i++){pT->CopyW(pT,&sP.wParam,&pH->byPassword[i*2]);FPUT(BOX_REG,pM);sP.byA2++;}sP.byA1++;} //5 KP Password
    if(pA->byA1==1){sP.byA2 = 0;for(i=0;i<8;i++){pT->CopyW(pT,&sP.wParam,&pH->byPhone0[i*2]);  FPUT(BOX_REG,pM);sP.byA2++;}sP.byA1++;} //6 Kp Phone 0
	if(pA->byA1==2){sP.byA2 = 0;for(i=0;i<8;i++){pT->CopyW(pT,&sP.wParam,&pH->byPhone1[i*2]);  FPUT(BOX_REG,pM);sP.byA2++;}sP.byA1++;} //7 Kp Phone 1
    if(pA->byA1==3){sP.byA2 = 0;for(i=0;i<8;i++){pT->CopyW(pT,&sP.wParam,&pH->byPhone2[i*2] ); FPUT(BOX_REG,pM);sP.byA2++;}sP.byA1++;} //8 Kp Phone 2

	if(pA->byA1==4){sP.byA2 = 0;sP.wParam = (WORD)pH->byKpID;      FPUT(BOX_REG,pM);sP.byA1++;}//0 Kp ID
	if(pA->byA1==5){sP.byA2 = 0;sP.wParam = (WORD)pH->byStoreMode; FPUT(BOX_REG,pM);sP.byA1++;}//1 Buffer Mode
	if(pA->byA1==6){sP.byA2 = 0;sP.wParam = (WORD)pH->byAmCall;    FPUT(BOX_REG,pM);sP.byA1++;}//2 Amout Call
	if(pA->byA1==7){sP.byA2 = 0;sP.wParam = (WORD)pH->byCallPeriod;FPUT(BOX_REG,pM);sP.byA1++;}//3 Call Period
	//if(pA->byA1==8){sP.byA2 = 0;sP.wParam = (WORD)pH->bySetChann;  FPUT(BOX_REG,pM);sP.byA1++;}//4 Call Period
    return FCHECK(BOX_REG);
}
BYTE CRegModule_CreatePortParam(This,SREGADDR *pA)
{
    DECLARE_SINGLE_OPEN(CRegModule)
	SREGPARAM sP;
	BYTE *pM = (BYTE*)&sP;
	SHARDCOMPUTERTABLE *pH = pT->m_pHCT;

	SARMINTERFACE *pR;
	BYTE byID = pA->byA1;
    sP.wSize  = sizeof(SREGPARAM);
	sP.byA0   = pA->byA0;
	sP.byA1   = pA->byA1;
	sP.byA2   = 0;
	if(byID<pH->byArmAmout)
	{
	 FFREE(BOX_REG);
	 pR = pH->pArmInterface[byID];
     sP.wParam = (WORD)pR->byNumber;         FPUT(BOX_REG,pM);sP.byA2++;  //0 Port Number
     sP.wParam = (WORD)pR->byType;           FPUT(BOX_REG,pM);sP.byA2++;  //1 Port Type
     sP.wParam = (WORD)pR->byPortRate;       FPUT(BOX_REG,pM);sP.byA2++;  //2 Port Type
     sP.wParam = (WORD)pR->stTcpAddr.byAddr0;FPUT(BOX_REG,pM);sP.byA2++;  //3 Parity
     sP.wParam = (WORD)pR->stTcpAddr.byAddr1;FPUT(BOX_REG,pM);sP.byA2++;  //4 Data Bits
     sP.wParam = (WORD)pR->stTcpAddr.byAddr2;FPUT(BOX_REG,pM);sP.byA2++;  //5 Stop Bits
	 return FCHECK(BOX_REG);
	}
	return 0;
}
BYTE CRegModule_CreateHardParam(This,SREGADDR *pA)
{
    DECLARE_SINGLE_OPEN(CRegModule)
	SREGPARAM sP;
	BYTE *pM = (BYTE*)&sP;
	SHARDCOMPUTERTABLE *pH = pT->m_pHCT;
	SHARDSLOT *pR;
	BYTE byID = pA->byA1;
    sP.wSize  = sizeof(SREGPARAM);
	sP.byA0   = pA->byA0;
	sP.byA1   = pA->byA1;
	sP.byA2   = 0;
	if(byID<pH->bySlotAmout)
	{
	 FFREE(BOX_REG);
	 pR = &pH->sSlot[byID];
	 sP.wParam = (WORD)pR->bySlotNumber;   FPUT(BOX_REG,pM);sP.byA2++; //0
	 sP.wParam = (WORD)pR->bySlotType;     FPUT(BOX_REG,pM);sP.byA2++; //1
	 sP.wParam = (WORD)pR->byPinAmout;     FPUT(BOX_REG,pM);sP.byA2++; //2
	 sP.wParam = (WORD)pR->byState;        FPUT(BOX_REG,pM);sP.byA2++; //3
	 sP.wParam = (WORD)pR->byAlmState;     FPUT(BOX_REG,pM);sP.byA2++; //4
	 return FCHECK(BOX_REG);
	}
    return 0;
}
BYTE CRegModule_CreateSoftTIParam(This,SREGADDR *pA)
{
    DECLARE_SINGLE_OPEN(CRegModule)
	SREGPARAM sP;
	BYTE *pM        = (BYTE*)&sP;
	SDIRTABLE *pD   = &pT->m_pSCT->sDirectionTable[0];
	BYTE byAmObject = pD->byAmSwitching;
	STIPARAM *pTI;
	BYTE byID = pA->byA1;
    sP.wSize  = sizeof(SREGPARAM);
	sP.byA0   = pA->byA0;
	sP.byA1   = pA->byA1;
	sP.byA2   = 0;
	sP.wParam = 0;
	if(pA->byA1<pD->byAmTI)
	{
 	 FFREE(BOX_REG);
     pTI = (STIPARAM*)pD->pSwitchTable[byID];
	 sP.wParam = (WORD)pTI->byID;          FPUT(BOX_REG,pM);sP.byA2++; //0
	 sP.wParam = (WORD)pTI->byAmParam;     FPUT(BOX_REG,pM);sP.byA2++; //1
	 sP.wParam = (WORD)pTI->byType;        FPUT(BOX_REG,pM);sP.byA2++; //2
	 sP.wParam = (WORD)pTI->bySlot;        FPUT(BOX_REG,pM);sP.byA2++; //3
	 sP.wParam = (WORD)pTI->byPin;         FPUT(BOX_REG,pM);sP.byA2++; //4
	 sP.wParam = (WORD)pTI->byAlmState;    FPUT(BOX_REG,pM);sP.byA2++; //5
	 sP.wParam = (WORD)pTI->byState;       FPUT(BOX_REG,pM);sP.byA2++; //6
	 sP.wParam = (WORD)pTI->byPriority;    FPUT(BOX_REG,pM);sP.byA2++; //7
	 sP.wParam = (WORD)pTI->byDrTimer;     FPUT(BOX_REG,pM);sP.byA2++; //8
	 sP.wParam = pTI->wHiLimit;            FPUT(BOX_REG,pM);sP.byA2++; //9
	 sP.wParam = pTI->wHiGister;           FPUT(BOX_REG,pM);sP.byA2++; //10
	 sP.wParam = pTI->wLoGister;           FPUT(BOX_REG,pM);sP.byA2++; //11
	 sP.wParam = pTI->wLoLimit;            FPUT(BOX_REG,pM);sP.byA2++; //12
	 sP.wParam = pTI->wLo;                 FPUT(BOX_REG,pM);sP.byA2++; //13
	 sP.wParam = pTI->wHi;                 FPUT(BOX_REG,pM);sP.byA2++; //14
	 sP.wParam = pTI->wEvPercent;          FPUT(BOX_REG,pM);sP.byA2++; //15
	 sP.wParam = pTI->wParam;              FPUT(BOX_REG,pM);sP.byA2++; //16
	 return FCHECK(BOX_REG);
	}
	return 0;
}
BYTE CRegModule_CreateSoftTSParam(This,SREGADDR *pA)
{
    DECLARE_SINGLE_OPEN(CRegModule)
	SREGPARAM sP;
	BYTE *pM        = (BYTE*)&sP;
	SDIRTABLE *pD   = &pT->m_pSCT->sDirectionTable[0];
	BYTE byAmObject = pD->byAmSwitching;
	STSPARAM *pTS;
	BYTE byID = pA->byA1+pD->byAmTI;
    sP.wSize  = sizeof(SREGPARAM);
	sP.byA0   = pA->byA0;
	sP.byA1   = pA->byA1;
	sP.byA2   = 0;
	sP.wParam = 0;
	if(pA->byA1<pD->byAmTS)
	{
 	 FFREE(BOX_REG);
	 pTS = (STSPARAM*)pD->pSwitchTable[byID];
	 sP.wParam = (WORD)pTS->byID;               FPUT(BOX_REG,pM);sP.byA2++; //0
	 sP.wParam = (WORD)pTS->byAmParam;          FPUT(BOX_REG,pM);sP.byA2++; //1
	 sP.wParam = (WORD)pTS->byType;		        FPUT(BOX_REG,pM);sP.byA2++; //2
	 sP.wParam = (WORD)pTS->bySlot;             FPUT(BOX_REG,pM);sP.byA2++; //3
	 sP.wParam = (WORD)pTS->byPin;              FPUT(BOX_REG,pM);sP.byA2++; //4
	 sP.wParam = (WORD)pTS->byAlmState;         FPUT(BOX_REG,pM);sP.byA2++; //5
     sP.wParam = (WORD)pTS->byState;            FPUT(BOX_REG,pM);sP.byA2++; //6
	 sP.wParam = (WORD)pTS->byPriority;         FPUT(BOX_REG,pM);sP.byA2++; //7
	 sP.wParam = (WORD)pTS->byCRemPulce;        FPUT(BOX_REG,pM);sP.byA2++; //8
	 sP.wParam = (WORD)pTS->byCSetPulce;        FPUT(BOX_REG,pM);sP.byA2++; //9
	 sP.wParam = (WORD)pTS->byAlarmMode;        FPUT(BOX_REG,pM);sP.byA2++; //10
	 sP.wParam = (WORD)pTS->byParam;            FPUT(BOX_REG,pM);sP.byA2++; //12
	 return FCHECK(BOX_REG);
	}
	return 0;
}
BYTE CRegModule_CreateSoftTUParam(This,SREGADDR *pA)
{
    DECLARE_SINGLE_OPEN(CRegModule)
	SREGPARAM sP;
	BYTE *pM        = (BYTE*)&sP;
	SDIRTABLE *pD   = &pT->m_pSCT->sDirectionTable[0];
	BYTE byAmObject = pD->byAmSwitching;
	STUPARAM *pTU;
	BYTE byID = pA->byA1+pD->byAmTI+pD->byAmTS;
    sP.wSize  = sizeof(SREGPARAM);
	sP.byA0   = pA->byA0;
	sP.byA1   = pA->byA1;
	sP.byA2   = 0;
	sP.wParam = 0;
	if(pA->byA1<pD->byAmTU)
	{
 	 FFREE(BOX_REG);
	 pTU = (STUPARAM*)pD->pSwitchTable[byID];
	 sP.wParam = (WORD)pTU->byID;              FPUT(BOX_REG,pM);sP.byA2++; //0
	 sP.wParam = (WORD)pTU->byAmParam;         FPUT(BOX_REG,pM);sP.byA2++; //1
	 sP.wParam = (WORD)pTU->byType;            FPUT(BOX_REG,pM);sP.byA2++; //2
	 sP.wParam = (WORD)pTU->bySlot;            FPUT(BOX_REG,pM);sP.byA2++; //3
	 sP.wParam = (WORD)pTU->byPin;             FPUT(BOX_REG,pM);sP.byA2++; //4
	 sP.wParam = (WORD)pTU->byAlmState;        FPUT(BOX_REG,pM);sP.byA2++; //5
	 sP.wParam = (WORD)pTU->byState;           FPUT(BOX_REG,pM);sP.byA2++; //6
	 sP.wParam = (WORD)pTU->byPulceType;       FPUT(BOX_REG,pM);sP.byA2++; //7
	 sP.wParam = (WORD)pTU->byCSetPulce;       FPUT(BOX_REG,pM);sP.byA2++; //8
	 sP.wParam = (WORD)pTU->byParam;           FPUT(BOX_REG,pM);sP.byA2++; //9
	 return FCHECK(BOX_REG);
	}
	return 0;
}
BYTE CRegModule_CreateSoftTRParam(This,SREGADDR *pA)
{
    DECLARE_SINGLE_OPEN(CRegModule)
	return 0;
}
BYTE CRegModule_SetKpParam(This,SREGPARAM *pA)
{
    DECLARE_SINGLE_OPEN(CRegModule)
    BYTE a1 = pA->byA1;
    BYTE a2 = pA->byA2;
	BYTE *pM = (BYTE*)pA;
	BYTE bySmode,byMask;
	SKPPARAM *pH   = pT->m_pHCT->pKpParam;
	if(a1==0) pT->CopyW(pT,&pH->byPassword[a2],&pA->wParam);else
	if(a1==1) pT->CopyW(pT,&pH->byPhone0[a2]  ,&pA->wParam);else
	if(a1==2) pT->CopyW(pT,&pH->byPhone1[a2]  ,&pA->wParam);else
	if(a1==3) pT->CopyW(pT,&pH->byPhone2[a2]  ,&pA->wParam);else
	if(a1==4) pH->byKpID       = (BYTE*)pA->wParam;
	if(a1==5)
	{
	 bySmode = (BYTE)pA->wParam;
	 byMask  = bySmode & 0x7f;
	 if(!(bySmode&0x80)) pH->byStoreMode |= byMask;
	 if(bySmode&0x80)    pH->byStoreMode &= ~byMask;
	}else
	if(a1==6) pH->byAmCall     = (BYTE)pA->wParam;else
	if(a1==7) pH->byCallPeriod = (BYTE)pA->wParam;else
	//if(a1==8) pH->bySetChann   = (BYTE)pA->wParam;else
	return 1;
}
BYTE CRegModule_SetPortParam(This,SREGPARAM *pA)
{
	DECLARE_SINGLE_OPEN(CRegModule)
	BYTE *pM = (BYTE*)pA;
	SHARDCOMPUTERTABLE *pH = pT->m_pHCT;
	SARMINTERFACE *pR;
	BYTE byID = pA->byA1;
	if(byID<pH->byArmAmout)
	{
	 pR = pH->pArmInterface[byID];
	 if(pA->byA2==0) pR->byNumber          = (BYTE)pA->wParam; //Port Number
	 if(pA->byA2==1) pR->byType            = (BYTE)pA->wParam; //Port Type
	 if(pA->byA2==2) pR->byPortRate        = (BYTE)pA->wParam; //Port Rate
	 if(pA->byA2==3) pR->stTcpAddr.byAddr0 = (BYTE)pA->wParam; //Parity
	 if(pA->byA2==4) pR->stTcpAddr.byAddr1 = (BYTE)pA->wParam; //Data Bits
	 if(pA->byA2==5) pR->stTcpAddr.byAddr2 = (BYTE)pA->wParam; //Stop Bits
	 return 1;
	}
	return 0;
}
BYTE CRegModule_SetHardParam(This,SREGPARAM *pA)
{
    DECLARE_SINGLE_OPEN(CRegModule)
	BYTE *pM = (BYTE*)pA;
	SHARDCOMPUTERTABLE *pH = pT->m_pHCT;
	SHARDSLOT *pR;
	BYTE byID = pA->byA1;
	if(byID<pH->bySlotAmout)
	{
	 pR = &pH->sSlot[byID];
	 if(pA->byA2==0) pR->bySlotNumber = (BYTE)pA->wParam;
     if(pA->byA2==1) pR->bySlotType   = (BYTE)pA->wParam;
	 if(pA->byA2==2) pR->byPinAmout   = (BYTE)pA->wParam;
	 if(pA->byA2==3) pR->byState      = (BYTE)pA->wParam;
	 if(pA->byA2==4) pR->byAlmState   = (BYTE)pA->wParam;
	 return 1;
	}
	return 0;
}
BYTE CRegModule_SetSoftTIParam(This,SREGPARAM *pA)
{
    DECLARE_SINGLE_OPEN(CRegModule)
	STIPARAM *pTI;
	SDIRTABLE *pD = &pT->m_pSCT->sDirectionTable[0];
	BYTE byID = pA->byA1;
	if(byID<pD->byAmSwitching)
	{
	 pTI = (STIPARAM*)pD->pSwitchTable[byID];
	 if(pA->byA2==0)  pTI->byID        = (BYTE)pA->wParam;
	 if(pA->byA2==1)  pTI->byAmParam   = (BYTE)pA->wParam;
	 if(pA->byA2==2)  pTI->byType      = (BYTE)pA->wParam;
	 if(pA->byA2==3)  pTI->bySlot      = (BYTE)pA->wParam;
	 if(pA->byA2==4)  pTI->byPin       = (BYTE)pA->wParam;
	 if(pA->byA2==5)  pTI->byAlmState  = (BYTE)pA->wParam;
	 if(pA->byA2==6)  pTI->byState     = (BYTE)pA->wParam;
	 if(pA->byA2==7)  pTI->byPriority  = (BYTE)pA->wParam;
	 if(pA->byA2==8) {pTI->byDrTimer   = (BYTE)pA->wParam;if(pTI->byDrTimer==0)pTI->byDrTimer=1;}
	 if(pA->byA2==9)  pTI->wHiLimit    = pA->wParam;
	 if(pA->byA2==10) pTI->wHiGister   = pA->wParam;
	 if(pA->byA2==11) pTI->wLoGister   = pA->wParam;
	 if(pA->byA2==12) pTI->wLoLimit    = pA->wParam;
	 if(pA->byA2==13) pTI->wLo         = pA->wParam;
	 if(pA->byA2==14) pTI->wHi         = pA->wParam;
	 if(pA->byA2==15) pTI->wEvPercent  = pA->wParam;
	 if(pA->byA2==16) pTI->wParam      = pA->wParam;
	 return 1;
	}
	return 0;
}
BYTE CRegModule_SetSoftTSParam(This,SREGPARAM *pA)
{
    DECLARE_SINGLE_OPEN(CRegModule)
	STSPARAM *pTS;
	SDIRTABLE *pD = &pT->m_pSCT->sDirectionTable[0];
	BYTE byID = pA->byA1+pD->byAmTI;
	if(byID<pD->byAmSwitching)
	{
	 pTS = (STSPARAM*)pD->pSwitchTable[byID];
	 if(pA->byA2==0)  pTS->byID        = (BYTE)pA->wParam;
	 if(pA->byA2==1)  pTS->byAmParam   = (BYTE)pA->wParam;
	 if(pA->byA2==2)  pTS->byType      = (BYTE)pA->wParam;
	 if(pA->byA2==3)  pTS->bySlot      = (BYTE)pA->wParam;
	 if(pA->byA2==4)  pTS->byPin       = (BYTE)pA->wParam;
	 if(pA->byA2==5)  pTS->byAlmState  = (BYTE)pA->wParam;
	 if(pA->byA2==6)  pTS->byState     = (BYTE)pA->wParam;
	 if(pA->byA2==7)  pTS->byPriority  = (BYTE)pA->wParam;
	 if(pA->byA2==8) {pTS->byCRemPulce = (BYTE)pA->wParam;if(pTS->byCRemPulce==0)pTS->byCRemPulce = 1;}
	 if(pA->byA2==9) {pTS->byCSetPulce = (BYTE)pA->wParam;if(pTS->byCSetPulce==0)pTS->byCSetPulce = 1;}
	 if(pA->byA2==10) pTS->byAlarmMode = (BYTE)pA->wParam;
	 if(pA->byA2==11) pTS->byParam     = (BYTE)pA->wParam;
	 return 1;
	}
	return 0;
}
BYTE CRegModule_SetSoftTUParam(This,SREGPARAM *pA)
{
    DECLARE_SINGLE_OPEN(CRegModule)
	STUPARAM *pTU;
	SDIRTABLE *pD = &pT->m_pSCT->sDirectionTable[0];
	BYTE byID = pA->byA1+pD->byAmTI+pD->byAmTS;
	if(byID<pD->byAmSwitching)
	{
	 pTU = (STUPARAM*)pD->pSwitchTable[byID];
	 if(pA->byA2==0)  pTU->byID        = (BYTE)pA->wParam;
	 if(pA->byA2==1)  pTU->byAmParam   = (BYTE)pA->wParam;
	 if(pA->byA2==2)  pTU->byType      = (BYTE)pA->wParam;
	 if(pA->byA2==3)  pTU->bySlot      = (BYTE)pA->wParam;
	 if(pA->byA2==4)  pTU->byPin       = (BYTE)pA->wParam;
	 if(pA->byA2==5)  pTU->byAlmState  = (BYTE)pA->wParam;
	 if(pA->byA2==6)  pTU->byState     = (BYTE)pA->wParam;
	 if(pA->byA2==7)  pTU->byPulceType = (BYTE)pA->wParam;
	 if(pA->byA2==8) {pTU->byCSetPulce = (BYTE)pA->wParam;if(pTU->byCSetPulce==0)pTU->byCSetPulce = 1;}
	 if(pA->byA2==9)  pTU->byParam     = (BYTE)pA->wParam;
	 return 1;
	}
	return 0;
}
BYTE CRegModule_SetSoftTRParam(This,SREGPARAM *pA)
{
    DECLARE_SINGLE_OPEN(CRegModule)
    return 0;
}
void CRegModule_CopyW(This,PVOID pvDst,PVOID pvSrc)
{
    DECLARE_SINGLE_OPEN(CRegModule)
	BYTE *pDS = (BYTE*)pvDst;
	BYTE *pSR = (BYTE*)pvSrc;
    #ifndef WIN32
	pDS[0] = pSR[1];
	pDS[1] = pSR[0];
    #else
	pDS[0] = pSR[0];
	pDS[1] = pSR[1];
    #endif
}
void CRegModule_CRegModule(This)
{
    DECLARE_SINGLE_OPEN(CRegModule)
	DECLARE_REGISTRATION(CRegModule,Init)
	DECLARE_REGISTRATION(CRegModule,QueryParam)
	DECLARE_REGISTRATION(CRegModule,SaveParam)
	DECLARE_REGISTRATION(CRegModule,CreateKpParam)
	DECLARE_REGISTRATION(CRegModule,CreatePortParam)
	DECLARE_REGISTRATION(CRegModule,CreateHardParam)
	DECLARE_REGISTRATION(CRegModule,CreateSoftTIParam)
	DECLARE_REGISTRATION(CRegModule,CreateSoftTSParam)
	DECLARE_REGISTRATION(CRegModule,CreateSoftTUParam)
	DECLARE_REGISTRATION(CRegModule,CreateSoftTRParam)

	DECLARE_REGISTRATION(CRegModule,SetKpParam)
	DECLARE_REGISTRATION(CRegModule,SetPortParam)
	DECLARE_REGISTRATION(CRegModule,SetHardParam)
	DECLARE_REGISTRATION(CRegModule,SetSoftTIParam)
	DECLARE_REGISTRATION(CRegModule,SetSoftTSParam)
	DECLARE_REGISTRATION(CRegModule,SetSoftTUParam)
	DECLARE_REGISTRATION(CRegModule,SetSoftTRParam)

	DECLARE_REGISTRATION(CRegModule,CopyW)
}
void CRegModule_DCRegModule(This)
{
	DECLARE_SINGLE_OPEN(CRegModule)
}
DECLARE_SINGLE_CREATE(CRegModule)
```

#### bnrsensr.c
```c
/********************************************************************
 * COPYRIGHT -- Kontora
 ********************************************************************
 * Program: bnrmain
 * File: bnrsensr.c
 * Author: Abramenya
 * Created: January 23, 2009
 *******************************************************************/
#include "bnrsensr.h"
#include "bnrdirmodule.h"
#if MYSYSTEM_ID != 5
SINT *chSensType[] =
{
	"SMART",
	"IDLES",
	"EMPTY"
};
SINT *chParType[] =
{
	"LEVEL",
	"TEMPR",
	"PRESS"
};
char *StateInfol[]  =
{
    "SNS_STATE_FREE",
};
char *ValInfol[]  =
{
	"INC_INP",
	"STATE",
};
void CSensor_Init(This,SSWITCHTABLE *pSTable)
{
    DECLARE_MULTI_OPEN(CSensor,CAuto)
	BYTE i;
	INT nS = sizeof(SNSPARAMTABLE);
	SNSPARAMTABLE *sP = (SNSPARAMTABLE*)pSTable->sSensorParamTable;
	COutGate *pG      = pT->m_pOutGate[0];
	pT->m_pvPT        = sP;
	pT->m_wSnsMode    = 0;
	pT->m_blSensorState = pSTable->blEnable;
	pT->m_pStateList   = pSTable->m_pStateList;
	pT->SetSensorID(pT,pSTable->bySensorID);
    memcpy(&pT->m_sPT,sP,sizeof(SNSPARAMTABLE));
	memcpy(&pT->m_sGT,pSTable->sOutGate[0],sizeof(SOUTGATE));
	strcpy(pT->m_sPT.m_chSNname,pG->m_chName);
	pT->m_sPT.m_swOpenTime = pG->m_wOTime;
	pT->m_sPT.m_sbyPmode   = pG->m_byMode;
	pT->m_sPT.m_sbyOmode   = pG->m_byOType;
	pT->m_sPT.m_srOmin     = pG->m_rMinRamp;
	pT->m_sPT.m_srOmax     = pG->m_rMaxRamp;
	pT->m_byPidMode        = pG->m_byMode;
	pG->SetMinRamp(pG,pT->m_sPT.m_srOmin);
	pG->SetMaxRamp(pG,pT->m_sPT.m_srOmax);
	pT->m_byParamType      = sP->m_sbyParamType;
	pT->m_bySensorType     = sP->m_snType;
	pT->m_bySwitchCommand  = pSTable->bySwitchCommand;
	if (pT->m_sPT.m_sbyInpState==ST_OPEN) pT->m_blInState  = TRUE; else pT->m_blInState   = FALSE;
	if ((pT->m_sPT.m_sbyOutState==ST_INIT)||(pT->m_sPT.m_sbyOutState==ST_CLOS))
	pT->m_blOutState = FALSE; else pT->m_blOutState = TRUE;
	pT->m_blProcState= TRUE;
	if (sP->m_sbyMode==SNS_MD_MANU) pT->SetManMode(pT);
	if (sP->m_sbyMode==SNS_MD_AUTO) pT->SetAutoMode(pT);
	if (sP->m_sbyMode==SNS_MD_LOOP) pT->SetLoopMode(pT);
	if(pT->m_bySensorType!=SNS_EMPTY)
	{
	 pT->CalcGate(pT);
	 if (!pT->m_blOutState)for (i=0;i<pT->m_byAmOutGate;i++)pT->m_pOutGate[i]->SetDefault(pT->m_pOutGate[i]);
	}
	pT->m_blStatState = FALSE;
	pT->m_wStatIndex  = 0;
	pT->m_wStatQuant  = 50;
	#ifdef DEB_CSensor
	//Info("\n(%b)CSSNS::>Create Sensor.Type:%s.",&pSTable->bySensorID,chSensType[pT->m_bySensorType]);
	#endif
	pT->m_blAlmLoLevel  = FALSE;
	pT->m_blRAlmLoLevel = FALSE;
	pT->m_blAlmHiLevel  = FALSE;
	pT->m_blRAlmHiLevel = FALSE;
	pT->m_blProcLoLevel = FALSE;
    pT->m_blProcHiLevel = FALSE;
	pT->m_dwAutoTime    = 0;
	pB->v[INC_INP]      = 0;
    pT->m_byAutoState   = SNS_STATE_FREE;
	pB->SetState(pB,SNS_STATE_FREE);
	pT->m_nInp->FilterEnable(pT->m_nInp,pT->m_sPT.m_byFilterOn);
  	pT->InitSensor(pC,sP);
	//pT->m_nInp = (INT16*)pT->m_pFCP->GetAddrPin(pT->m_pFCP->pChld);
	/*
	InitObject(CMTimer,&pT->m_nATmr[TMR_SET_ALM_HI]);
	InitObject(CMTimer,&pT->m_nATmr[TMR_REM_ALM_HI]);
	InitObject(CMTimer,&pT->m_nATmr[TMR_SET_ALM_LO]);
	InitObject(CMTimer,&pT->m_nATmr[TMR_REM_ALM_LO]);
	pT->m_nATmr[TMR_SET_ALM_HI].SetTimer(&pT->m_nATmr[TMR_SET_ALM_HI],MDL_SENSR,MDL_SENSR,EV_SENSR_TMR_SAHI+TMR_SET_ALM_HI,pT->m_byDirection,pT->m_bySensorID,DEV_SYSTM_BOX_ID);
	pT->m_nATmr[TMR_REM_ALM_HI].SetTimer(&pT->m_nATmr[TMR_REM_ALM_HI],MDL_SENSR,MDL_SENSR,EV_SENSR_TMR_SAHI+TMR_REM_ALM_HI,pT->m_byDirection,pT->m_bySensorID,DEV_SYSTM_BOX_ID);
	pT->m_nATmr[TMR_SET_ALM_LO].SetTimer(&pT->m_nATmr[TMR_SET_ALM_LO],MDL_SENSR,MDL_SENSR,EV_SENSR_TMR_SAHI+TMR_SET_ALM_LO,pT->m_byDirection,pT->m_bySensorID,DEV_SYSTM_BOX_ID);
	pT->m_nATmr[TMR_REM_ALM_LO].SetTimer(&pT->m_nATmr[TMR_REM_ALM_LO],MDL_SENSR,MDL_SENSR,EV_SENSR_TMR_SAHI+TMR_REM_ALM_LO,pT->m_byDirection,pT->m_bySensorID,DEV_SYSTM_BOX_ID);
	*/
}
void CSensor_InitDigital(This,SSWITCHTABLE *pSTable)
{
    DECLARE_MULTI_OPEN(CSensor,CAuto)
	pT->m_pStateList = pSTable->m_pStateList;
	pB->SetState(pB,SNS_STATE_FREE);
	pT->SetSensorID(pT,pSTable->bySensorID);
    pT->m_bySwitchCommand = pSTable->bySwitchCommand;
	pT->SetAutoMode(pT);
	pT->InitSensor(pC,pSTable);
}
void CSensor_SetOutState(This,BYTE byState)
{
    DECLARE_MULTI_OPEN(CSensor,CAuto)
	BYTE i;
    if ((byState==ST_INIT)||(byState==ST_CLOS)) pT->m_blOutState = FALSE; else pT->m_blOutState = TRUE;
	for (i=0;i<pT->m_byAmOutGate;i++)
    pT->m_pOutGate[i]->SetState(pT->m_pOutGate[i],byState);
	pT->m_sPT.m_sbyOutState = byState;
}
void CSensor_CalcGate(This)
{
    DECLARE_MULTI_OPEN(CSensor,CAuto)
	pT->m_nAcpMin     = ACP_MIN;
	pT->m_nAcpMax     = ACP_MAX;
	pT->m_iHiLimit    = pT->m_nAcpMax;
	pT->m_iLoLimit    = pT->m_nAcpMin;
	pT->m_iPHiLimit   = pT->GetInParam(pT,pT->m_sPT.m_swHiOper);
	pT->m_iPLoLimit   = pT->GetInParam(pT,pT->m_sPT.m_swLoOper);
	pT->m_iHiAlmLimit = pT->GetInParam(pT,pT->m_sPT.m_swHiAlLimit);
	pT->m_iLoAlmLimit = pT->GetInParam(pT,pT->m_sPT.m_swLoAlLimit);
	pT->m_nIniValue   = pT->GetInParam(pT,pT->m_sPT.m_swInitValue);
	pT->m_iIPLoLimit  = pT->m_iPLoLimit;
	pT->m_iIPHiLimit  = pT->m_iPHiLimit;
	if(pT->m_byPidMode==SINV)
	{
     pT->m_iPHiLimit   = pT->m_nAcpMax - pT->m_iPHiLimit;
	 pT->m_iLoLimit    = pT->m_nAcpMax - pT->m_iLoLimit;
	 pT->m_iHiAlmLimit = pT->m_nAcpMax - pT->m_iHiAlmLimit;
	 pT->m_iLoAlmLimit = pT->m_nAcpMax - pT->m_iLoAlmLimit;
	 pT->m_nIniValue   = pT->m_nAcpMax - pT->m_nIniValue;
	}
    #ifdef MY_MODEL
	if(pT->m_byPidMode==SDIR)
	{
	 pT->m_nInPin = (UINT)(REAL)(pT->m_nIniValue)/pT->m_nInp->m_rKoef;
	 pT->m_nInp->SetInput(pT->m_nInp,pT->m_nInPin);
	}
    #endif
}
void CSensor_InitSensor(This,SNSPARAMTABLE *pParam)
{
	DECLARE_MULTI_OPEN(CSensor,CAuto)
    pT->m_blInState   = FALSE;
	pT->m_blProcState = FALSE;
	pT->m_blOutState  = FALSE;
	pT->m_nInPin      = -1;
	pT->m_nOutPin     = -1;
}
void CSensor_GetParamTable(This,BYTE byOwner)
{
    DECLARE_MULTI_OPEN(CSensor,CAuto)
	SNSPARAMTABLE psT;
	SHMESSAGE m_sMsg;
	COutGate *pG = pT->m_pOutGate[0];
    m_sMsg.m_sbyFrom      = MDL_DIRMD;
	m_sMsg.m_sbyFor       = byOwner;
	m_sMsg.m_sbyIntType   = DEV_ARM_PORT_TCP;
	m_sMsg.m_sbyType      = EV_SENSR_GET_SNPARAM_IND;
	m_sMsg.m_sbyServerID  = pT->m_bySystemID;
	m_sMsg.m_sbyDirection = pT->m_byDirection;
	m_sMsg.m_sbySensor    = pT->m_bySensorID;
    m_sMsg.m_sbyInfo[0]   = 1+sizeof(SNSPARAMTABLE);
	m_sMsg.m_swLen        = 9+m_sMsg.m_sbyInfo[0];
	psT.m_swResistance    = pT->GetRealParam(pT,(BYTE*)&pT->m_sPT.m_swResistance);
	psT.m_swHiLimit       = pT->GetRealParam(pT,(BYTE*)&pT->m_sPT.m_swHiLimit);
	psT.m_swLoLimit       = pT->GetRealParam(pT,(BYTE*)&pT->m_sPT.m_swLoLimit);
	psT.m_swHiAlLimit     = pT->GetRealParam(pT,(BYTE*)&pT->m_sPT.m_swHiAlLimit);
	psT.m_swLoAlLimit     = pT->GetRealParam(pT,(BYTE*)&pT->m_sPT.m_swLoAlLimit);
	psT.m_swHiOper        = pT->GetRealParam(pT,(BYTE*)&pT->m_sPT.m_swHiOper);
	psT.m_swLoOper        = pT->GetRealParam(pT,(BYTE*)&pT->m_sPT.m_swLoOper);
	psT.m_swInitValue     = pT->GetRealParam(pT,(BYTE*)&pT->m_sPT.m_swInitValue);
	psT.m_swMaxAcpInp     = pT->GetWordParam(pT,(BYTE*)&pT->m_sPT.m_swMaxAcpInp);
	psT.m_swMaxAcpOut     = pT->GetWordParam(pT,(BYTE*)&pT->m_sPT.m_swMaxAcpOut);
	psT.m_swOpenTime      = pT->GetWordParam(pT,(BYTE*)&pT->m_sPT.m_swOpenTime);
	//psT.m_swPidDiffMode   = pT->GetWordParam(pT,(BYTE*)&pT->m_sPT.m_swPidDiffMode);
	psT.bySrcSlotNumber   = pT->m_sPT.bySrcSlotNumber;
	psT.m_swPidDiffMode   = pT->m_sPT.m_swPidDiffMode;
	psT.m_snType          = pT->m_sPT.m_snType;
	psT.m_sbyParamType    = pT->m_sPT.m_sbyParamType;
	psT.m_sbyInpState     = pT->m_sPT.m_sbyInpState;
	psT.m_sbyOutState     = pT->m_sPT.m_sbyOutState;
	if (byOwner==MDL_ARMSY) psT.m_sbyOutState = pG->GetPrcGate(pG);
	psT.m_sbyMode         = pT->m_sPT.m_sbyMode;
	psT.m_snType          = pT->m_sPT.m_snType;
	psT.m_byFilterOn      = pT->m_sPT.m_byFilterOn;
	psT.m_sbyPmode        = pT->m_sPT.m_sbyPmode;
	psT.m_sbyOmode        = pT->m_sPT.m_sbyOmode;
	psT.m_srOmin          = pT->GetRealParam(pT,(BYTE*)&pT->m_sPT.m_srOmin);
	psT.m_srOmax          = pT->GetRealParam(pT,(BYTE*)&pT->m_sPT.m_srOmax);

	strcpy(psT.m_chSNname,pT->m_sPT.m_chSNname);
    memcpy(&m_sMsg.m_sbyInfo[1],&psT,sizeof(SNSPARAMTABLE));
    FPUT(DEV_ARMOT_BOX_ID,(BYTE*)&m_sMsg);
	pT->GetParam(pC,byOwner);
}
void CSensor_SEventHandler(This,SMESSAGE *pMsg)
{
	DECLARE_MULTI_OPEN(CSensor,CAuto)
	BYTE byLen,byInitType,byPType,byPLen,i,byGate,byValue;
	REAL rlPrcOpen;
	COutGate *pG;
	INT16 wParam;
	UINT nParam;
	REAL rParam;
	switch(pMsg->m_sbyType)
	{
	  case EV_SENSR_TMR_SAHI:
	  case EV_SENSR_TMR_RAHI:
	  case EV_SENSR_TMR_SALO:
	  case EV_SENSR_TMR_RALO:
		   pT->SetMsgAuto(pT,pMsg);
	  break;
      case EV_SMSNS_SET_PARAM_REQ:
		   byLen      = pMsg->m_sbyInfo[0];
		   byInitType = pMsg->m_sbyInfo[1];
		   byPType    = pMsg->m_sbyInfo[2];
		   byPLen     = pMsg->m_sbyInfo[3];
           #ifdef DEB_CSensor
		   Info("\n(%b)CSNSR::>DC(%b,%b)SSP:%M.",&pT->m_bySystemID,&pT->m_byDirection,&pT->m_bySensorID,(BYTE*)pMsg);
           #endif
		   if(byInitType==SNS_SENS_INI)
		   {
		   switch(byPType)
		   {
		    case PR_Out_En:
		         pT->m_sPT.m_sbyOutState = pMsg->m_sbyInfo[4];
		         if(pT->m_sPT.m_sbyOutState==ST_INIT)
				 {
		          for (i=0;i<pT->m_byAmOutGate;i++)pT->m_pOutGate[i]->SetDefault(pT->m_pOutGate[i]);
		          pT->m_blOutState = FALSE;
				 }
		         if(pT->m_sPT.m_sbyOutState==ST_OPEN)
				 {
		          for (i=0;i<pT->m_byAmOutGate;i++)pT->m_pOutGate[i]->SetState(pT->m_pOutGate[i],ST_OPEN);
		          pT->m_blOutState = TRUE;
				 }
		    break;
		    case PR_LO:
			     rParam = pT->GetRealParam(pT,&pMsg->m_sbyInfo[4]);
			     pT->m_sPT.m_swLoLimit = rParam;
			     pT->m_iLoLimit        = pT->RealToAcp(pT,pT->m_sPT.m_swLoLimit);
		    break;
			case PR_HI:
                 rParam =  pT->GetRealParam(pT,&pMsg->m_sbyInfo[4]);
			     pT->m_sPT.m_swHiLimit = rParam;
			     pT->m_iHiLimit        = pT->RealToAcp(pT,pT->m_sPT.m_swHiLimit);
		    break;
			case PR_ALO:
			     rParam =  pT->GetRealParam(pT,&pMsg->m_sbyInfo[4]);
			     pT->m_sPT.m_swLoAlLimit = rParam;
			     pT->m_iLoAlmLimit       = pT->RealToAcp(pT,pT->m_sPT.m_swLoAlLimit);
		    break;
			case PR_AHI:
			     rParam =  pT->GetRealParam(pT,&pMsg->m_sbyInfo[4]);
			     pT->m_sPT.m_swHiAlLimit = rParam;
			     pT->m_iHiAlmLimit       = pT->RealToAcp(pT,pT->m_sPT.m_swHiAlLimit);
		    break;
			case PR_PHI:
			     rParam = pT->GetRealParam(pT,&pMsg->m_sbyInfo[4]);
			     nParam = pT->RealToAcp(pT,rParam);
				 if ((rParam>=pT->m_sPT.m_swLoOper)&&(rParam<=pT->m_sPT.m_swHiAlLimit))
				 {
			      if(pT->m_byParamType==P_PRESS)pT->SetForAll(pT,P_PRESS,PR_PHI,rParam,nParam);else
				  {
				   pT->m_iIPHiLimit     = nParam;
				   if(pT->m_byPidMode==SINV) nParam = pT->m_iHiLimit - nParam;
				   pT->m_iPHiLimit      = nParam;
			       pT->m_sPT.m_swHiOper = rParam;
				  }
				 }
		    break;
			case PR_PLO:
			     rParam = pT->GetRealParam(pT,&pMsg->m_sbyInfo[4]);
			     nParam = pT->RealToAcp(pT,rParam);
				 if ((rParam<=pT->m_sPT.m_swHiOper)&&(rParam>=pT->m_sPT.m_swLoAlLimit))
				 {
			      if(pT->m_byParamType==P_PRESS)pT->SetForAll(pT,P_PRESS,PR_PLO,rParam,nParam);else
				  {
				   pT->m_iIPLoLimit     = nParam;
				   if(pT->m_byPidMode==SINV) nParam = pT->m_iHiLimit - nParam;
 				   pT->m_iPLoLimit      = nParam;
			       pT->m_sPT.m_swLoOper = rParam;
				  }
				 }
		    break;
		    case PR_ACO:
		 	     pT->m_sPT.m_swMaxAcpInp  = pT->GetWordParam(pT,&pMsg->m_sbyInfo[4]);
			     pT->m_pOutGate[0]->m_wBase = pT->m_sPT.m_swMaxAcpInp;
		    break;
			case PR_ACM:
				 pT->m_sPT.m_swMaxAcpOut  = pT->GetWordParam(pT,&pMsg->m_sbyInfo[4]);
				 pT->m_nAcpOutRamp        = pT->m_sPT.m_swMaxAcpOut;
			break;
			case PR_OTIME:
				 pT->m_sPT.m_swOpenTime   = pT->GetWordParam(pT,&pMsg->m_sbyInfo[4]);
				 pT->m_sGT.wOpenTime      = pT->m_sPT.m_swOpenTime;
				 pG = pT->m_pOutGate[0];
			     if(pG)pG->SetOutTime(pG,pT->m_sPT.m_swOpenTime);
            break;
		    case PR_RST:
			     pT->m_sPT.m_swResistance = pT->GetRealParam(pT,&pMsg->m_sbyInfo[4]);
				 pT->m_nInp->SetResistance(pT->m_nInp,pT->m_sPT.m_swResistance);
		    break;
		    case PR_INI:
			     pT->m_sPT.m_swInitValue  = pT->GetRealParam(pT,&pMsg->m_sbyInfo[4]);
		    break;
            case PR_X:
			     pT->EventHandler(pC,pMsg);
		    break;
		    case PR_out_mode:
			     if(pMsg->m_sbyInfo[4]==0) pT->SetManMode(pT);
		         if(pMsg->m_sbyInfo[4]==1) pT->SetAutoMode(pT);
			     if(pMsg->m_sbyInfo[4]==2) pT->SetLoopMode(pT);
			     pT->EventHandler(pC,pMsg);
		    break;
		    case PR_INC_IN:
				 wParam = pT->GetWordParam(pT,&pMsg->m_sbyInfo[4]);
				 pT->IncInput(pC,wParam);
		    break;
			case PR_EnFlt:
			     pT->m_sPT.m_byFilterOn = pMsg->m_sbyInfo[4];
				 pT->m_nInp->FilterEnable(pT->m_nInp,pT->m_sPT.m_byFilterOn);
			break;
		    default:
		    break;
		   }
		   }
		   if(byInitType==SNS_SENS_CTR)
		   {
		   switch(byPType)
		   {
		    case PR_OPN_GT:
			     byGate    = pMsg->m_sbyInfo[4];
			     rlPrcOpen = pT->GetRealParam(pT,&pMsg->m_sbyInfo[5]);
			     pT->m_bySensorID = pT->m_bySensorID;
                 if(pT->m_sPT.m_sbyMode==SNS_MD_MANU)
				 {
			      pG = pT->m_pOutGate[byGate];
			      if(pG)pG->OpenGate(pG,rlPrcOpen);
				 }
			break;
			case PR_STOP_GT:
				 byGate    = pMsg->m_sbyInfo[4];
				 if(pT->m_sPT.m_sbyMode==SNS_MD_MANU)
				 {
				  pG = pT->m_pOutGate[byGate];
				  if(pG)pG->StopGate(pG);
				 }
			break;
			case PR_PRC_GT:
                 byGate    = pMsg->m_sbyInfo[4];
				 byValue   = pMsg->m_sbyInfo[5];
				 if(pT->m_sPT.m_sbyMode==SNS_MD_MANU)
				 {
				  pG = pT->m_pOutGate[byGate];
				  if(pG)pG->OpenGateReq(pG,byValue);
				 }
			break;
		    default:
            break;
		   }
		   }
		   if(byInitType==SNS_SENS_OUT)
		   {
		   switch(byPType)
		   {
		    case PR_OMIN:
			     pT->m_sPT.m_srOmin = pT->GetRealParam(pT,&pMsg->m_sbyInfo[4]);
			     pT->m_sGT.rMinRamp = pT->m_sPT.m_srOmin;
			     pT->m_pOutGate[0]->SetMinRamp(pT->m_pOutGate[0],pT->m_sPT.m_srOmin);
				 pT->EventHandler(pC,pMsg);
			break;
			case PR_OMAX:
			     pT->m_sPT.m_srOmax = pT->GetRealParam(pT,&pMsg->m_sbyInfo[4]);
			     pT->m_sGT.rMaxRamp = pT->m_sPT.m_srOmax;
			     pT->m_pOutGate[0]->SetMaxRamp(pT->m_pOutGate[0],pT->m_sPT.m_srOmax);
				 pT->EventHandler(pC,pMsg);
			break;
			case PR_PMODE:
			     pT->m_sPT.m_sbyPmode = pMsg->m_sbyInfo[4];
			     pT->m_sGT.byMode = pT->m_sPT.m_sbyPmode;
			     pT->m_pOutGate[0]->m_byMode = pT->m_sPT.m_sbyPmode;
			     memcpy(&pT->m_sPT,pT->m_pvPT,sizeof(SNSPARAMTABLE));
			     strcpy(pT->m_sPT.m_chSNname,pT->m_pOutGate[0]->m_chName);
			     pT->m_sPT.m_sbyPmode = pT->m_pOutGate[0]->m_byMode;
			     pT->m_sPT.m_sbyOmode = pT->m_pOutGate[0]->m_byOType;
			     pT->m_sPT.m_srOmin   = pT->m_pOutGate[0]->m_rMinRamp;
			     pT->m_sPT.m_srOmax   = pT->m_pOutGate[0]->m_rMaxRamp;
			     pT->m_byPidMode      = pT->m_pOutGate[0]->m_byMode;
			     pT->CalcGate(pT);
			break;
			case PR_OMODE:
			     pT->m_sPT.m_sbyOmode = pMsg->m_sbyInfo[4];
			     pT->m_sGT.byOType = pT->m_sPT.m_sbyOmode;
		  	     pT->m_pOutGate[0]->m_byOType = pT->m_sPT.m_sbyOmode;
			break;
			default:
			break;
		   }
		   }
	  break;
	  default:
      break;
	}
}
void CSensor_SetForAll(This,BYTE byPType,BYTE byPCode,REAL rParam,UINT nParam)
{
	DECLARE_MULTI_OPEN(CSensor,CAuto)
	BYTE i;
	CSensor *p;
	DWORD dwSet = 0;
	CDirectionModule *pDR = (CDirectionModule*)pT->m_pvDirection;
	BYTE byAmSens = pDR->m_byAmSwitching;
	if((pT->m_bySystemID==3)&&(pT->m_bySensorID==2))dwSet = 0x0c;else
	if((pT->m_bySystemID!=3)&&(pT->m_bySensorID==0))dwSet = 0x03;else
	if((pT->m_bySystemID!=3)&&(pT->m_bySensorID==2))dwSet = 0x0c;else
	dwSet |= 1<<pT->m_bySensorID;
	for (i=0;i<byAmSens;i++)
	{
	 p = pDR->m_pSensor[i];
	 if(p->m_byParamType==byPType)
	 {
	  if(dwSet&(1<<i))
	  {
	   if(byPCode==PR_PLO) p->m_iIPLoLimit = nParam;
	   if(byPCode==PR_PHI) p->m_iIPHiLimit = nParam;
	   if(p->m_byPidMode==SINV)
	   {
	    nParam = p->m_iHiLimit - nParam;
	   }
	   if(byPCode==PR_PLO)
	   {
		p->m_iPLoLimit = nParam;
		p->m_sPT.m_swLoOper = rParam;
	   }
	   if(byPCode==PR_PHI)
	   {
		p->m_iPHiLimit = nParam;
		p->m_sPT.m_swHiOper = rParam;
	   }
	  }
	 }
	}
}
void CSensor_SetLEMode(This)
{
	DECLARE_MULTI_OPEN(CSensor,CAuto)
}
void CSensor_IncInput(This,INT16 wParam)
{
    DECLARE_MULTI_OPEN(CSensor,CAuto)
}
INT16 CSensor_GetWordParam(This,BYTE *pbyParam)
{
    DECLARE_MULTI_OPEN(CSensor,CAuto)
	INT16 wValue;
	BYTE *pBT = (BYTE*)&wValue;
    #ifndef WIN32
	pBT[0] = pbyParam[1];
	pBT[1] = pbyParam[0];
    #else
	pBT[0] = pbyParam[0];
	pBT[1] = pbyParam[1];
    #endif
	return wValue;
}
REAL CSensor_GetRealParam(This,BYTE *pbyParam)
{
    DECLARE_MULTI_OPEN(CSensor,CAuto)
	REAL rlValue;
	BYTE *pR = (BYTE*)&rlValue;
    #ifndef WIN32
	pR[3] = pbyParam[0];
	pR[2] = pbyParam[1];
	pR[1] = pbyParam[2];
	pR[0] = pbyParam[3];
    #else
	memcpy(&rlValue,pbyParam,4);
	#endif
	return rlValue;
}
UINT CSensor_GetInParam(This,REAL nParam)
{
    DECLARE_MULTI_OPEN(CSensor,CAuto)
	REAL k;
	REAL rnParam  = nParam;
    REAL rnAcpMin = (REAL)pT->m_nAcpMin;
	REAL rnAcpMax = (REAL)pT->m_nAcpMax;
	REAL rnParamMax = pT->m_sPT.m_swHiLimit;
	k = rnParamMax/(rnAcpMax-rnAcpMin);
    return (UINT)(rnParam/k+rnAcpMin);
}
UINT CSensor_AcpToInt(This,UINT nAcpCode)
{
	DECLARE_MULTI_OPEN(CSensor,CAuto)
	REAL k;
    REAL rnAcpMin   = (REAL)pT->m_nAcpMin;
	REAL rnAcpMax   = (REAL)pT->m_nAcpMax;
	REAL rnParamMax = (REAL)pT->m_sPT.m_swHiLimit;
	REAL rnAcpCode  = (REAL)nAcpCode;
	k = rnParamMax/(rnAcpMax-rnAcpMin);
    return (UINT)((rnAcpCode-rnAcpMin)*k);
}
UINT CSensor_IntToAcp(This,UINT nParam)
{
	DECLARE_MULTI_OPEN(CSensor,CAuto)
	REAL k;
	REAL rnParam    = (REAL)nParam;
    REAL rnAcpMin   = (REAL)pT->m_nAcpMin;
	REAL rnAcpMax   = (REAL)pT->m_nAcpMax;
	REAL rnParamMax = (REAL)pT->m_sPT.m_swHiLimit;
	k = rnParamMax/(rnAcpMax-rnAcpMin);
    return (UINT)(rnParam/k+rnAcpMin);
}
REAL CSensor_AcpToReal(This,UINT nAcpCode)
{
	DECLARE_MULTI_OPEN(CSensor,CAuto)
	REAL k;
    REAL rnAcpMin   = (REAL)pT->m_nAcpMin;
	REAL rnAcpMax   = (REAL)pT->m_nAcpMax;
	REAL rnParamMax = (REAL)pT->m_sPT.m_swHiLimit;
	REAL rnAcpCode  = (REAL)nAcpCode;
	k = rnParamMax/(rnAcpMax-rnAcpMin);
    return (rnAcpCode-rnAcpMin)*k;
}
UINT CSensor_RealToAcp(This,REAL nParam)
{
	DECLARE_MULTI_OPEN(CSensor,CAuto)
	REAL k;
	REAL rnParam    = nParam;
    REAL rnAcpMin   = (REAL)pT->m_nAcpMin;
	REAL rnAcpMax   = (REAL)pT->m_nAcpMax;
	REAL rnParamMax = (REAL)pT->m_sPT.m_swHiLimit;
	k = rnParamMax/(rnAcpMax-rnAcpMin);
    return (UINT)(rnParam/k+rnAcpMin);
}
void CSensor_GetParam(This,BYTE byParam)
{
	DECLARE_MULTI_OPEN(CSensor,CAuto)
}
void CSensor_SetLoopMode(This)
{
	DECLARE_MULTI_OPEN(CSensor,CAuto)
	pT->m_sPT.m_sbyMode   = SNS_MD_LOOP;
    #ifdef DEB_CSensor
	Info("\n(%b)CSNSR::>DC(%b,%b)SET:SNS_MD_LOOP.",&pT->m_bySystemID,&pT->m_byDirection,&pT->m_bySensorID);
    #endif
}
void CSensor_SetManMode(This)
{
	DECLARE_MULTI_OPEN(CSensor,CAuto)
	CDirectionModule *pDR = (CDirectionModule*)pT->m_pvDirection;
	pT->EnableInput(pT,FALSE);
	pT->EnableProc(pT,FALSE);
	pT->EnableOutput(pT,FALSE);
	pT->m_sPT.m_sbyMode = SNS_MD_MANU;
	pDR->m_wSensorMode &= ~(1<<pT->m_bySensorID);
	pT->Serialize(pC,TRUE);
    #ifdef DEB_CSensor
	Info("\n(%b)CSNSR::>DC(%b,%b)SET:SNS_MD_MANU.",&pT->m_bySystemID,&pT->m_byDirection,&pT->m_bySensorID);
    #endif
}
void CSensor_SetAutoMode(This)
{
	DECLARE_MULTI_OPEN(CSensor,CAuto)
	CDirectionModule *pDR = (CDirectionModule*)pT->m_pvDirection;
	pT->EnableInput(pT,TRUE);
	pT->EnableProc(pT,TRUE);
	pT->EnableOutput(pT,TRUE);
	pT->m_sPT.m_sbyMode = SNS_MD_AUTO;
	pDR->m_wSensorMode |= 1<<pT->m_bySensorID;
	pT->Serialize(pC,FALSE);
    #ifdef DEB_CSensor
	Info("\n(%b)CSNSR::>DC(%b,%b)SET:SNS_MD_AUTO.",&pT->m_bySystemID,&pT->m_byDirection,&pT->m_bySensorID);
    #endif
}
void CSensor_Serialize(This,BOOL byDir){}
INT16** CSensor_GetCaptureBuffer(This)
{
    DECLARE_MULTI_OPEN(CSensor,CAuto)
	return (INT16**)pT->m_pwStatBuff;
}
void CSensor_StartCaptureProc(This)
{
    DECLARE_MULTI_OPEN(CSensor,CAuto)
	pT->m_blStatState = TRUE;
	pT->m_wStatIndex  = 0;
	pT->m_wStatQuant  = 50;
}
void CSensor_StopCaptureProc(This)
{
    DECLARE_MULTI_OPEN(CSensor,CAuto)
	pT->m_blStatState = FALSE;
}
void CSensor_RestartCaptureProc(This)
{
    DECLARE_MULTI_OPEN(CSensor,CAuto)
	pT->m_blStatState = TRUE;
	pT->m_wStatIndex  = 0;
}
void CSensor_CaptureData(This){}
void CSensor_OpenGate(This)
{
    DECLARE_MULTI_OPEN(CSensor,CAuto)
	pT->m_wStatIndex = 0;
	pT->m_blCaptureState = TRUE;
}
void CSensor_CloseGate(This)
{
    DECLARE_MULTI_OPEN(CSensor,CAuto)
	pT->m_blCaptureState = FALSE;
}
void CSensor_AddData(This,DINT dData)
{
    DECLARE_MULTI_OPEN(CSensor,CAuto)
	BYTE *pWT;
    #ifndef WIN32
	BYTE *pWS;
    #endif
	if (pT->m_blCaptureState)
	{
	 pWT = (BYTE*)&pT->m_pwStatBuff[pT->m_wStatIndex++];
     #ifndef WIN32
	 pWS = (BYTE*)&dData;
	 pWT[3] = pWS[0];
	 pWT[2] = pWS[1];
	 pWT[1] = pWS[2];
	 pWT[0] = pWS[3];
     #else
	 memcpy(pWT,&dData,4);
     #endif
	}
}
void CSensor_AddCaptureData(This,DINT nP0,DINT nP1,DINT nP2)
{
    DECLARE_MULTI_OPEN(CSensor,CAuto)
	BYTE *pWT;
    #ifndef WIN32
	BYTE *pWS;
    #endif
	if(pT->m_blStatState)
	{
		pWT = (BYTE*)&pT->m_pwStatBuff[pT->m_wStatIndex++];
		#ifndef WIN32
		pWS = (BYTE*)&nP0;
		pWT[3] = pWS[0];
		pWT[2] = pWS[1];
		pWT[1] = pWS[2];
		pWT[0] = pWS[3];
        #else
        memcpy(pWT,&nP0,4);
		#endif
		pWT = (BYTE*)&pT->m_pwStatBuff[pT->m_wStatIndex++];
        #ifndef WIN32
		pWS = (BYTE*)&nP1;
		pWT[3] = pWS[0];
		pWT[2] = pWS[1];
		pWT[1] = pWS[2];
		pWT[0] = pWS[3];
        #else
        memcpy(pWT,&nP1,4);
        #endif
		pWT = (BYTE*)&pT->m_pwStatBuff[pT->m_wStatIndex++];
        #ifndef WIN32
		pWS = (BYTE*)&nP2;
		pWT[3] = pWS[0];
		pWT[2] = pWS[1];
		pWT[1] = pWS[2];
		pWT[0] = pWS[3];
        #else
        memcpy(pWT,&nP2,4);
        #endif
	 if(pT->m_wStatIndex==3*pT->m_wStatQuant)
	 pT->m_blStatState = FALSE;
	}
}
void CSensor_StopStatProc(This)
{
    DECLARE_MULTI_OPEN(CSensor,CAuto)
	pT->m_blStatState = TRUE;
}
void CSensor_EnableInput(This,BOOL blState)
{
	DECLARE_MULTI_OPEN(CSensor,CAuto)
	pT->m_blInState = blState;
	//Info("\n(%b)CHAND::>EnableInput:%b",&pT->m_bySensorID,&pT->m_blInState);
}
void CSensor_EnableProc(This,BOOL blState)
{
	DECLARE_MULTI_OPEN(CSensor,CAuto)
	pT->m_blProcState = blState;
	//Info("\n(%b)CHAND::>EnableProc:%b",&pT->m_bySensorID,&pT->m_blProcState);
}
void CSensor_EnableOutput(This,BOOL blState)
{
	DECLARE_MULTI_OPEN(CSensor,CAuto)
	pT->m_blOutState = blState;
	//Info("\n(%b)CHAND::>EnableOutput:%b",&pT->m_bySensorID,&pT->m_blOutState);
}
void CSensor_SetParType(This,BYTE byParType)
{
	DECLARE_MULTI_OPEN(CSensor,CAuto)
	pT->m_byParamType = byParType;
}
BYTE CSensor_GetParType(This)
{
    DECLARE_MULTI_OPEN(CSensor,CAuto)
	return pT->m_byParamType;
}
void CSensor_SetSensorID(This,BYTE bySensID)
{
    DECLARE_MULTI_OPEN(CSensor,CAuto)
	pT->m_bySensorID = bySensID;
}
BYTE CSensor_GetSensorID(This)
{
    DECLARE_MULTI_OPEN(CSensor,CAuto)
	return pT->m_bySensorID;
}
BYTE CSensor_GetDirection(This)
{
    DECLARE_MULTI_OPEN(CSensor,CAuto)
	return pT->m_byDirection;
}
void CSensor_SetDirection(This,PVOID pvDir,BYTE byDir)
{
    DECLARE_MULTI_OPEN(CSensor,CAuto)
    pT->m_byDirection = byDir;
	pT->m_pvDirection = pvDir;
}
void CSensor_ObserveProc(This)
{
	DECLARE_MULTI_OPEN(CSensor,CAuto)
	if(pT->m_blInState)   pT->PreProc(pC);
	if(pT->m_blProcState) pT->Processing(pC);
	if(pT->m_blOutState)  pT->PostProc(pC);
    pT->RunAutomat(pC);
}
void CSensor_RunAutomat(This)
{
	DECLARE_MULTI_OPEN(CSensor,CAuto)
}
void CSensor_EventGen(This)
{
    DECLARE_MULTI_OPEN(CSensor,CAuto)
	UINT uVL  = (UINT)pT->m_nInPin;
	UINT uHIA = pT->m_iHiAlmLimit;
	UINT uLOA = pT->m_iLoAlmLimit;
    UINT uPHI = pT->m_iPHiLimit;
	UINT uPLO = pT->m_iPLoLimit;
    UINT Hi   = pT->m_nAcpMax;
	UINT Lo   = pT->m_nAcpMin;
	if(pT->m_byPidMode==SINV)
	{
	 uVL  = Hi-(UINT)pT->m_nInPin;
	 uHIA = Hi-pT->m_iHiAlmLimit;
	 uLOA = Hi-pT->m_iLoAlmLimit;
     uPHI = Hi-pT->m_iPHiLimit;
	 uPLO = Hi-pT->m_iPLoLimit;
	}
	if((uVL>=Lo)&&(uVL<uLOA))  pT->SetEvent(pT,&pT->m_blAlmLoLevel ,&pT->m_blRAlmLoLevel,EV_ADMIN_SET_ALM_LOLEV_REQ);
	else pT->SetEvent(pT,&pT->m_blRAlmLoLevel,&pT->m_blAlmLoLevel ,EV_ADMIN_REM_ALM_LOLEV_REQ);//Lo Alarm
    if((uVL>uLOA)&&(uVL<uPLO))pT->SetEvent(pT,&pT->m_blProcLoLevel,&pT->m_blProcHiLevel,EV_ADMIN_OPER_LO_REQ);//Proced
    if((uVL>uPHI)&&(uVL<Hi))  pT->SetEvent(pT,&pT->m_blProcHiLevel,&pT->m_blProcLoLevel,EV_ADMIN_OPER_HI_REQ);//Proced
    if((uVL>=uHIA)&&(uVL<=Hi))  pT->SetEvent(pT,&pT->m_blAlmHiLevel ,&pT->m_blRAlmHiLevel,EV_ADMIN_SET_ALM_HILEV_REQ);
	else pT->SetEvent(pT,&pT->m_blRAlmHiLevel,&pT->m_blAlmHiLevel ,EV_ADMIN_REM_ALM_HILEV_REQ);//Li Alarm
}
void CSensor_SetEvent(This,BOOL *bl0,BOOL *bl1,BYTE byEvent)
{
    DECLARE_MULTI_OPEN(CSensor,CAuto)
	if (*bl0 == FALSE)
	{
	 //Info("\n(%b)CSNSR[%b]::>SEND:EV[%b].",&pT->m_bySystemID,&pT->m_bySensorID,&byEvent);
	 pB->HandleEvent(pB,byEvent);
     *bl0 = TRUE;
     *bl1 = FALSE;
	}
}
void CSensor_ConnectFCP(This,CInputGate *pInputGate)
{
    DECLARE_MULTI_OPEN(CSensor,CAuto)
	pT->m_nInp = pInputGate;
}
void CSensor_ConnectOutGate(This,COutGate *pOGate)
{
    DECLARE_MULTI_OPEN(CSensor,CAuto)
	BYTE byID = pOGate->m_byGateID;
    pT->m_pOutGate[byID] = pOGate;
}
void CSensor_SetLoLimit(This,UINT iValue)
{
    DECLARE_MULTI_OPEN(CSensor,CAuto)
	pT->m_iPLoLimit = iValue;
}
void CSensor_SetHiLimit(This,UINT iValue)
{
    DECLARE_MULTI_OPEN(CSensor,CAuto)
	pT->m_iPHiLimit  = iValue;
	pT->m_iIPHiLimit = iValue;
}
///////////////////////
void CSensor_SetLoAlLimit(This,INT16 iValue)
{
    DECLARE_MULTI_OPEN(CSensor,CAuto)
	pT->m_iLoAlmLimit = iValue;
}
void CSensor_SetHiAlLimit(This,INT16 iValue)
{
    DECLARE_MULTI_OPEN(CSensor,CAuto)
	pT->m_iHiAlmLimit = iValue;
}
void CSensor_SetCallBackProc(This,PCLB pfCallBack)
{
	DECLARE_MULTI_OPEN(CSensor,CAuto)
	pT->m_pfnCallBackProc = pfCallBack;
}
void CSensor_SetState(This,DWORD dwState)
{
	DECLARE_MULTI_OPEN(CSensor,CAuto)
	pT->m_dwState = dwState;
}
DWORD CSensor_GetState(This)
{
	DECLARE_MULTI_OPEN(CSensor,CAuto)
	return pT->m_dwState;
}
void CSensor_Enable(This)
{
    DECLARE_MULTI_OPEN(CSensor,CAuto)
	pT->SetState(pT,ST01_SNS_OPEN);
}
void CSensor_Disable(This)
{
	DECLARE_MULTI_OPEN(CSensor,CAuto)
	pT->SetState(pT,ST02_SNS_CLOS);
}
void CSensor_PreProc(This)
{
    DECLARE_MULTI_OPEN(CSensor,CAuto)
}
void CSensor_Processing(This)
{
    DECLARE_MULTI_OPEN(CSensor,CAuto)
}
void CSensor_PostProc(This)
{
    DECLARE_MULTI_OPEN(CSensor,CAuto)
}
void CSensor_EventGate(This,BYTE byEvent)
{
    DECLARE_MULTI_OPEN(CSensor,CAuto)
}
void CSensor_ConnectPinAddres(This)
{
    DECLARE_MULTI_OPEN(CSensor,CAuto)
	BYTE i;
	CPin *pPN;
    for (i=0;i<pT->m_wAmInput;i++)
	{
     pPN = pT->m_pINP[i];
	 if(pPN->m_byPinType==PIN_AN_INOT_INT) pT->m_nINP[i] = pPN->GetAddrPin(pPN->pChld);
	 if(pPN->m_byPinType==PIN_DG_INOT_BOL) pT->m_bINP[i] = pPN->GetAddrPin(pPN->pChld);
	}
    for (i=0;i<pT->m_wAmOutput;i++)
	{
	 pPN = pT->m_pOUT[i];
	 if(pPN->m_byPinType==PIN_AN_INOT_INT) pT->m_nOUT[i] = pPN->GetAddrPin(pPN->pChld);
	 if(pPN->m_byPinType==PIN_DG_INOT_BOL) pT->m_bOUT[i] = pPN->GetAddrPin(pPN->pChld);
	}
}
void CSensor_SendCommand(This,BYTE byFor,BYTE byType)
{
    DECLARE_MULTI_OPEN(CSensor,CAuto)
	SHORTMESSAGE sMsg;
    sMsg.m_swLen        = 9;
	sMsg.m_sbyFrom      = MDL_SSENS;
    sMsg.m_sbyFor       = byFor;
	sMsg.m_sbyIntType   = DEV_SYS_INTERFACE;
	sMsg.m_sbyServerID  = pT->m_bySystemID;
	sMsg.m_sbyType      = byType;
	sMsg.m_sbyDirection = pT->m_byDirection;
	sMsg.m_sbySensor    = pT->m_bySensorID;
	FPUT(DEV_ADMIN_BOX_ID,(BYTE*)&sMsg);
}
//Auto Section
BOOL CSensor_HandleTask(This,TTask* pTask)
{
    DECLARE_MULTI_OPEN(CSensor,CAuto)
	COutGate *pG;
	BYTE V0,V1;
    for(;*pTask!=EXIT_D;pTask++)
    {
	  switch (*pTask)
	  {
	  	 case CMD_OPENGATE:
			  V0 = *(++pTask);
			  V1 = *(++pTask);
			  pG = pT->m_pOutGate[V0];
			  if(pG)pG->OpenGate(pG,V1);
              #ifdef DEB_CSensor
			  Info("\n(%b)CSNSR[%b]::>GATE:[%b]am[%b]",&pT->m_bySystemID,&pT->m_bySensorID,&V0,&V1);
              #endif
         break;
	  	 case CMD_SETSTATE:
			  V1 = *(++pTask);
			  if(*pTask==STATE) V1 = pB->v[STATE];
			  pB->SetState(pB,V1);
              #ifdef DEB_CSensor
			  Info("\n(%b)CSNSR[%b]::>STAT:%s->%s ",&pT->m_bySystemID,&pT->m_bySensorID,StateInfol[pB->v[STATE]],StateInfol[V1]);
			  //Info("\n(%b)CSNSR[%b]::>STAT:/--------New--------/",&pT->m_bySystemID,&pT->m_bySensorID);
              #endif
			  pB->v[STATE] = V1;
         break;
		 case CMD_SEND:
			  V0 = *(++pTask);
			  V1 = *(++pTask);
			  pT->SendCommand(pT,V0,V1);
              #ifdef DEB_CSensor
			  Info("\n(%b)CSNSR[%b]::>SEND:[%b][%b].",&pT->m_bySystemID,&pT->m_bySensorID,&V0,&V1);
              #endif
		 break;
		 case CMD_SETVALUE:
			  V0 = *(++pTask);
			  pB->v[V0] = *(++pTask);
              #ifdef DEB_CSensor
			  Info("\n(%b)CSNSR[%b]::>SETV:%s=%b",&pT->m_bySystemID,&pT->m_bySensorID,ValInfol[V0],&pB->v[V0]);
              #endif
		 break;
		 case CMD_TIMERON:
			  V0 = *(++pTask);//Timer ID
			  V1 = *(++pTask);//Time
			  pT->m_nATmr[V0].OnTimer(&pT->m_nATmr[V0],V1);
              #ifdef DEB_CSensor
			  Info("\n(%b)CSNSR[%b]::>TMON:[%b][%b].",&pT->m_bySystemID,&pT->m_bySensorID,&V0,&V1);
	          #endif
		 break;
		 case CMD_TIMEROFF:
			  V0 = *(++pTask);
			  pT->m_nATmr[V0].OfTimer(&pT->m_nATmr[V0]);
              #ifdef DEB_CSensor
			  Info("\n(%b)CSNSR[%b]::>TMOF:[%b].",&pT->m_bySystemID,&pT->m_bySensorID,&V0);
              #endif
		 break;
		 default:
		 break;
	  };
	}
	return TRUE;
}
TStateList* CSensor_GetStateList(This)
{
    DECLARE_MULTI_OPEN(CSensor,CAuto)
	return pT->m_pStateList;
}
void CSensor_SetMsgAuto(This,SMESSAGE *pMsg)
{
    DECLARE_MULTI_OPEN(CSensor,CAuto)
	BYTE byEvent = pMsg->m_sbyType;
	pB->HandleEvent(pB,byEvent);
}
void CSensor_SetAutoEvent(This,BYTE byEvent)
{
    DECLARE_MULTI_OPEN(CSensor,CAuto)
    pB->HandleEvent(pB,byEvent);
}
void CSensor_CSensor(This)
{
	DECLARE_MULTI_OPEN(CSensor,CAuto)
	BYTE i;
    DECLARE_REGISTRATION(CSensor,Init)
	DECLARE_REGISTRATION(CSensor,SetCallBackProc)
	DECLARE_REGISTRATION(CSensor,ObserveProc)
	DECLARE_REGISTRATION(CSensor,SetState)
	DECLARE_REGISTRATION(CSensor,GetState)
	DECLARE_REGISTRATION(CSensor,Enable)
	DECLARE_REGISTRATION(CSensor,Disable)
	DECLARE_REGISTRATION(CSensor,Init)
	DECLARE_REGISTRATION(CSensor,ConnectFCP)
	DECLARE_REGISTRATION(CSensor,SetLoLimit)
	DECLARE_REGISTRATION(CSensor,SetHiLimit)
	DECLARE_REGISTRATION(CSensor,SetLoAlLimit)
	DECLARE_REGISTRATION(CSensor,SetHiAlLimit)
	DECLARE_REGISTRATION(CSensor,SendCommand)

	DECLARE_REGISTRATION(CSensor,PreProc)
	DECLARE_REGISTRATION(CSensor,Processing)
	DECLARE_REGISTRATION(CSensor,PostProc)
	DECLARE_REGISTRATION(CSensor,SetDirection)
	DECLARE_REGISTRATION(CSensor,GetDirection)
	DECLARE_REGISTRATION(CSensor,SetSensorID)
	DECLARE_REGISTRATION(CSensor,GetSensorID)

	DECLARE_REGISTRATION(CSensor,SetParType)
	DECLARE_REGISTRATION(CSensor,GetParType)

	DECLARE_REGISTRATION(CSensor,EnableInput)
	DECLARE_REGISTRATION(CSensor,EnableProc)
	DECLARE_REGISTRATION(CSensor,EnableOutput)

	DECLARE_REGISTRATION(CSensor,SetLoopMode)
	DECLARE_REGISTRATION(CSensor,SetManMode)
	DECLARE_REGISTRATION(CSensor,SetAutoMode)
	//Statistic
	DECLARE_REGISTRATION(CSensor,StartCaptureProc)
	DECLARE_REGISTRATION(CSensor,StopCaptureProc)
	DECLARE_REGISTRATION(CSensor,AddCaptureData)
	DECLARE_REGISTRATION(CSensor,CaptureData)
	DECLARE_REGISTRATION(CSensor,RestartCaptureProc)
	DECLARE_REGISTRATION(CSensor,GetCaptureBuffer)
	DECLARE_REGISTRATION(CSensor,AddData)
	DECLARE_REGISTRATION(CSensor,OpenGate)
	DECLARE_REGISTRATION(CSensor,CloseGate)
	DECLARE_REGISTRATION(CSensor,GetParamTable)
	DECLARE_REGISTRATION(CSensor,GetParam)
	DECLARE_REGISTRATION(CSensor,SEventHandler)
	DECLARE_REGISTRATION(CSensor,GetWordParam)
	DECLARE_REGISTRATION(CSensor,GetRealParam)
	DECLARE_REGISTRATION(CSensor,InitSensor)
	DECLARE_REGISTRATION(CSensor,IncInput)
	DECLARE_REGISTRATION(CSensor,GetInParam)
	DECLARE_REGISTRATION(CSensor,CalcGate)
	DECLARE_REGISTRATION(CSensor,AcpToInt)
	DECLARE_REGISTRATION(CSensor,IntToAcp)
	DECLARE_REGISTRATION(CSensor,AcpToReal)
	DECLARE_REGISTRATION(CSensor,RealToAcp)
	DECLARE_REGISTRATION(CSensor,ConnectOutGate)
	DECLARE_REGISTRATION(CSensor,EventGen)

	DECLARE_REGISTRATION(CSensor,EventGate)
	DECLARE_REGISTRATION(CSensor,SetOutState)
	DECLARE_REGISTRATION(CSensor,RunAutomat)
	DECLARE_REGISTRATION(CSensor,SetForAll)
	DECLARE_REGISTRATION(CSensor,SetEvent)
	DECLARE_REGISTRATION(CSensor,RunAutomat)
	DECLARE_REGISTRATION(CSensor,InitDigital)
	DECLARE_REGISTRATION(CSensor,ConnectPinAddres)
	//Automat
	DECLARE_REGISTRATION(CSensor,SetMsgAuto)
	DECLARE_REGISTRATION(CSensor,SetAutoEvent)
	DECLARE_REGISTRATION(CSensor,Serialize)

	DECLARE_VIRTUAL_FUNC(CSensor,HandleTask)
	DECLARE_VIRTUAL_FUNC(CSensor,GetStateList)
    for(i=0;i<DEV_AMT_GATE_SNS;i++) pT->m_pOutGate[i] = 0;
	pT->m_pfnCallBackProc = NULL;
	pT->m_byEvent = 0xff;
	pT->m_dwState = ST02_SNS_CLOS;
	pT->m_nAcpMin = 6552;
	pT->m_nAcpMax = 32760;
}
void CSensor_DCSensor(This)
{
	DECLARE_MULTI_OPEN(CSensor,CAuto)
	BYTE i;
    for (i=0;i<pT->m_byAmOutGate;i++)
    DestroyObject(COutGate,pT->m_pOutGate[i]);
}
DECLARE_MULTI_CREATE(CSensor,CAuto)
#endif
```

#### bnrslide.c
```c
/********************************************************************
 * COPYRIGHT -- Kontora
 ********************************************************************
 * Program: bnrmain
 * File: bnrlsens.c
 * Author: Abramenya
 * Created: January 19, 2009
 *******************************************************************/

#include "bnrslide.h"
#ifdef _DEFAULT_INCLUDES
 #include <AsDefault.h>
#endif
void CSlot_Init(This,SHARDSLOT *psvSlot)
{
     DECLARE_SINGLE_OPEN(CSlot)
	 pT->m_bySlotNumber = psvSlot->bySlotNumber;
	 pT->m_bySlotType   = psvSlot->bySlotType;
	 pT->m_byAmPin      = psvSlot->byPinAmout;
	 pT->m_byState      = psvSlot->byState;
	 pT->m_pvAlmState   = psvSlot->pvAlmState;
	 pT->InitSlot(pC,psvSlot);
}
void CSlot_InitSlot(This,SHARDSLOT *psvSlot)
{
     DECLARE_SINGLE_OPEN(CSlot)
}
//Constructor-Destructor
void CSlot_CSlot(This)
{
     DECLARE_SINGLE_OPEN(CSlot)
	 DECLARE_REGISTRATION(CSlot,Init)
	 DECLARE_REGISTRATION(CSlot,InitSlot)
}
void CSlot_DCSlot(This)
{
	 DECLARE_SINGLE_OPEN(CSlot)
}
DECLARE_SINGLE_CREATE(CSlot)
```
